Universal Robots PolyScope program: elton_fulltask.urp

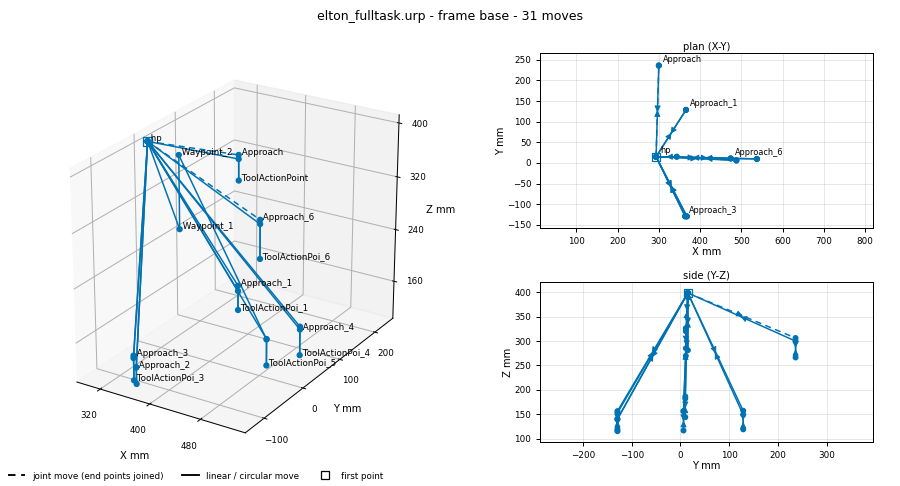
[picture p0: tool path of elton_fulltask.urp in frame base, 31 of 31 moves have a stored position in this frame; points joined in program order, loops and branches not executed]
Program elton_fulltask (installation=default directory=/programs createdIn=5.11.5.1010327 lastSavedIn=5.11.9.1010452 robotSerialNumber=20225200364)
Calibrated DH parameters: a=[0.00002, -0.569483, -0.54992, -0.00001, -0.000036, 0]; d=[0.180894, -146.691669, 192.918669, -46.053088, 0.119778, 0.115602]; alpha=[1.571425, -0.001534, 0.003359, 1.568739, -1.571477, 0]; deltaTheta=[0, 0.376258, -0.101074, -0.275185, -0.000002, 0]
Robot Program (runOnlyOnce=false)
  MoveL speed 250 mm/s, acceleration 1200 mm/s^2 (useActiveTCP=true) feature=Base
    Waypoint hp: TCP in base x=292.997 y=15.071 z=398.72 mm, rx=2.2312 ry=-2.2053 rz=0.0033 rad; joints [39.465, -75.549, -131.57, -243.154, -90.002, -141.049] deg
    URCap RG Grip (OnRobot, OnRobot A/S) dataModel(rg-target-force=40.0, rg-target-width=0.1)
    Loop Counting (count=6) loopVariable(name=Loop_2)
      URCap Palletizing (polyscope-pallet-impl, Universal Robots) dataModel(palletFeature=Base, isPalletizing=true, Length(key=objectHeight value=0.00001 unit=M), Variable(key=globalCountingVariable, variable(name=Pallet_4_cnt, initializeExpression=1)), Variable(key=layerNumberVariable, variable(name=Pallet_4_lno, initializeExpression=1)), Variable(key=layerCountingVariable, variable(name=Pallet_4_lct, initializeExpression=1)), Variable(key=handleSeparatorVariable, variable(name=Pallet_4_sep, initializeExpression=False)), Variable(key=totalCountVariable, variable(name=Pallet_4_tct, initializeExpression=1)), Variable(key=name, variable(name=R)), Variable(key=referencePoint, variable(featureName=referencePoin_3)), Variable(key=separatorPoint, variable(featureName=separatorPoin_3))); state(isChildrenLocked=true)
        URCap Patterns (polyscope-pallet-impl, Universal Robots) state(isChildrenLocked=true)
          URCap Pattern (polyscope-pallet-impl, Universal Robots) dataModel(UUID=4bae607c-6a0e-463c-838a-ad417c079e18, patternType=LINE, objects=6, Variable(key=nameVariable, variable(name=Line_Pattern_5))); state(isChildrenLocked=true)
            URCap Item (polyscope-pallet-impl, Universal Robots) dataModel(UUID=7363f219-9633-4242-9e50-65c058707edd, patternType=LINE, index=0, calibrationDeltaTheta=[-7.716858584048969E-7, 0.5809325624761351, 5.982441805008871, -0.2801932900558549, -2.087699179323388E-6, 7.182941588051994E-8], calibrationA=[5.584882619731399E-5, -0.5116748572506173, -0.549032347835167, 8.201669770320986E-5, -3.0447895639691726E-5, 0.0], calibrationD=[0.18058730552743416, -182.578946596082, 231.39006605348337, -48.6373829503458, 0.11974176219014578, 0.11553881708205978], calibrationAlpha=[1.5714381462339815, -0.001839843720035074, 0.003236774450590588, 1.5698364982897774, -1.571354041521518, 0.0], calibrationJointChecksum=[-1488423315, -1488334884, 658253144, -1490959501, -1490992896, -1492776484], calibrationStatus=2, calibrationValidChecksum=true, baseToFeature=[0.0, 0.0, 0.0, 0.0, 0.0, 0.0], TCPOffset=[-1.927819047531365E-5, -7.340324279514476E-6, -7.641604901187371E-6, 8.402270385809591E-6, 1.306011648505891E-6, 3.5749922966518936E-6], Variable(key=variable, variable(name=StartItem_5)), JointPositions(key=jointpositions, JointPosition(key=[1], Angle(key=pos value=1.151373 unit=RAD)), JointPosition(key=[2], Angle(key=pos value=-1.661465 unit=RAD)), JointPosition(key=[3], Angle(key=pos value=-2.268619 unit=RAD)), JointPosition(key=[4], Angle(key=pos value=-3.927088 unit=RAD)), JointPosition(key=[5], Angle(key=pos value=-1.572545 unit=RAD)), JointPosition(key=[6], Angle(key=pos value=-1.977698 unit=RAD))))
            URCap Item (polyscope-pallet-impl, Universal Robots) dataModel(UUID=34e06e1b-5aee-467a-bdea-27d33826544a, patternType=LINE, index=1, calibrationDeltaTheta=[-7.716858584048969E-7, 0.5809325624761351, 5.982441805008871, -0.2801932900558549, -2.087699179323388E-6, 7.182941588051994E-8], calibrationA=[5.584882619731399E-5, -0.5116748572506173, -0.549032347835167, 8.201669770320986E-5, -3.0447895639691726E-5, 0.0], calibrationD=[0.18058730552743416, -182.578946596082, 231.39006605348337, -48.6373829503458, 0.11974176219014578, 0.11553881708205978], calibrationAlpha=[1.5714381462339815, -0.001839843720035074, 0.003236774450590588, 1.5698364982897774, -1.571354041521518, 0.0], calibrationJointChecksum=[-1488423315, -1488334884, 658253144, -1490959501, -1490992896, -1492776484], calibrationStatus=2, calibrationValidChecksum=true, baseToFeature=[0.0, 0.0, 0.0, 0.0, 0.0, 0.0], TCPOffset=[-1.4484733942277117E-5, 2.1892267797196663E-6, -8.963613490398092E-6, 1.4148497921052897E-5, -4.324978428417448E-5, -3.9434016187655385E-5], Variable(key=variable, variable(name=EndItem_5)), JointPositions(key=jointpositions, JointPosition(key=[1], Angle(key=pos value=1.582831 unit=RAD)), JointPosition(key=[2], Angle(key=pos value=-1.495539 unit=RAD)), JointPosition(key=[3], Angle(key=pos value=-2.436687 unit=RAD)), JointPosition(key=[4], Angle(key=pos value=-3.925245 unit=RAD)), JointPosition(key=[5], Angle(key=pos value=-1.57402 unit=RAD)), JointPosition(key=[6], Angle(key=pos value=-1.546403 unit=RAD))))
        URCap Layers (polyscope-pallet-impl, Universal Robots) dataModel(separators=[false], selectedPatterns=[4bae607c-6a0e-463c-838a-ad417c079e18])
        URCap At Each Item (polyscope-pallet-impl, Universal Robots) dataModel(selectedPattern=4bae607c-6a0e-463c-838a-ad417c079e18, selectedPosition=7363f219-9633-4242-9e50-65c058707edd, Approach_calibrationDeltaTheta=[1.8465908720177726E-7, 0.2347954391419265, 6.32563174757166, -0.2772392005664852, -1.1261302130722607E-6, 2.5749233771577007E-7], Approach_calibrationA=[4.883734728215554E-5, -0.5955365338115801, -0.5495804852909227, 2.1882318399536237E-5, -4.077691201947169E-5, 0.0], Approach_calibrationD=[0.18075383087768818, -173.5375957069896, 228.42940994299985, -54.71797068756973, 0.11978402921182532, 0.11553172182396411], Approach_calibrationAlpha=[1.5713803919023464, -8.208946844426788E-4, 0.002849148556013, 1.569345144561223, -1.571367981038201, 0.0], Approach_calibrationJointChecksum=[-1454342380, -1456026624, 660707710, -1491716883, -1491592869, -1491595829], Approach_calibrationStatus=2, Approach_calibrationValidChecksum=true, Approach_baseToFeature=[0.0, 0.0, 0.0, 0.0, 0.0, 0.0], Approach_TCPOffset=[5.4603109008871664E-5, 2.376683340771235E-5, 1.3810152235949058E-5, -3.879481254340057E-5, 1.22456475810181E-4, -2.4036645708755116E-5], Exit_calibrationDeltaTheta=[1.8465908720177726E-7, 0.2347954391419265, 6.32563174757166, -0.2772392005664852, -1.1261302130722607E-6, 2.5749233771577007E-7], Exit_calibrationA=[4.883734728215554E-5, -0.5955365338115801, -0.5495804852909227, 2.1882318399536237E-5, -4.077691201947169E-5, 0.0], Exit_calibrationD=[0.18075383087768818, -173.5375957069896, 228.42940994299985, -54.71797068756973, 0.11978402921182532, 0.11553172182396411], Exit_calibrationAlpha=[1.5713803919023464, -8.208946844426788E-4, 0.002849148556013, 1.569345144561223, -1.571367981038201, 0.0], Exit_calibrationJointChecksum=[-1454342380, -1456026624, 660707710, -1491716883, -1491592869, -1491595829], Exit_calibrationStatus=2, Exit_calibrationValidChecksum=true, Exit_baseToFeature=[0.0, 0.0, 0.0, 0.0, 0.0, 0.0], Exit_TCPOffset=[5.458817584649833E-5, 2.1432463847392835E-5, 7.349381505572516E-5, -1.2814573171777247E-4, 1.0172603500468313E-4, -1.732072415206431E-5], currentWizardState=LANDING, Pose(key=refBaseToFeature, Position(key=posePosition, Length(key=X value=0 unit=M), Length(key=Y value=0 unit=M), Length(key=Z value=0 unit=M)), Rotation(key=poseRotation, Angle(key=RX value=0 unit=RAD), Angle(key=RY value=0 unit=RAD), Angle(key=RZ value=0 unit=RAD))), Pose(key=refPose, Position(key=posePosition, Length(key=X value=0.299651 unit=M), Length(key=Y value=0.236166 unit=M), Length(key=Z value=0.266297 unit=M)), Rotation(key=poseRotation, Angle(key=RX value=2.247176 unit=RAD), Angle(key=RY value=-2.190564 unit=RAD), Angle(key=RZ value=0.005192 unit=RAD))), JointPositions(key=Approach_jointpositions, JointPosition(key=[1], Angle(key=pos value=1.142609 unit=RAD)), JointPosition(key=[2], Angle(key=pos value=-1.611972 unit=RAD)), JointPosition(key=[3], Angle(key=pos value=-2.237967 unit=RAD)), JointPosition(key=[4], Angle(key=pos value=-4.008917 unit=RAD)), JointPosition(key=[5], Angle(key=pos value=-1.570991 unit=RAD)), JointPosition(key=[6], Angle(key=pos value=-2.021054 unit=RAD))), JointPositions(key=Exit_jointpositions, JointPosition(key=[1], Angle(key=pos value=1.142618 unit=RAD)), JointPosition(key=[2], Angle(key=pos value=-1.620563 unit=RAD)), JointPosition(key=[3], Angle(key=pos value=-2.243419 unit=RAD)), JointPosition(key=[4], Angle(key=pos value=-3.994874 unit=RAD)), JointPosition(key=[5], Angle(key=pos value=-1.570968 unit=RAD)), JointPosition(key=[6], Angle(key=pos value=-2.021008 unit=RAD))))
          URCap Generated Movements (polyscope-pallet-impl, Universal Robots) state(isChildrenLocked=true)
            MoveJ speed 60 deg/s, acceleration 80 deg/s^2 (useActiveTCP=true) feature=referencePoin_3
              Waypoint Approach: TCP in base x=299.628 y=236.111 z=306.226 mm, rx=2.2471 ry=-2.1905 rz=0.0053 rad; joints [65.467, -92.357, -128.232, -229.697, -90.01, -115.799] deg; TCP offset x=0 y=0 z=0 mm, rx=0 ry=0 rz=0 rad; feature pose in base x=299.651 y=236.166 z=266.297 mm, rx=2.2472 ry=-2.1906 rz=0.0052 rad
            MoveL speed 250 mm/s, acceleration 1200 mm/s^2 (useActiveTCP=true) feature(featureName=referencePoin_3)
              Waypoint ToolActionPoint: TCP in base x=299.651 y=236.166 z=266.297 mm, rx=2.2472 ry=-2.1906 rz=0.0052 rad; joints [65.47, -95.65, -130.086, -224.543, -90.002, -115.781] deg; TCP offset x=0 y=0 z=0 mm, rx=0 ry=0 rz=0 rad
            Folder Tool action
              URCap RG Grip (OnRobot, OnRobot A/S) dataModel(rg-target-force=40.0, rg-target-width=0.073)
            MoveL speed 250 mm/s, acceleration 1200 mm/s^2 (useActiveTCP=true) feature(featureName=referencePoin_3)
              Waypoint Exit_1: TCP in base x=299.631 y=236.111 z=299.866 mm, rx=2.2471 ry=-2.1904 rz=0.0052 rad; joints [65.465, -92.855, -128.546, -228.886, -90.014, -115.798] deg; TCP offset x=0 y=0 z=0 mm, rx=0 ry=0 rz=0 rad
      Waypoint hp: TCP in base x=292.997 y=15.071 z=398.72 mm, rx=2.2312 ry=-2.2053 rz=0.0033 rad; joints [39.465, -75.549, -131.57, -243.154, -90.002, -141.049] deg
      URCap Palletizing (polyscope-pallet-impl, Universal Robots) dataModel(palletFeature=Base, isPalletizing=true, Length(key=objectHeight value=0.00001 unit=M), Variable(key=globalCountingVariable, variable(name=Pallet_5_cnt, initializeExpression=1)), Variable(key=layerNumberVariable, variable(name=Pallet_5_lno, initializeExpression=1)), Variable(key=layerCountingVariable, variable(name=Pallet_5_lct, initializeExpression=1)), Variable(key=handleSeparatorVariable, variable(name=Pallet_5_sep, initializeExpression=False)), Variable(key=totalCountVariable, variable(name=Pallet_5_tct, initializeExpression=1)), Variable(key=name, variable(name=R2M)), Variable(key=referencePoint, variable(featureName=referencePoin_4)), Variable(key=separatorPoint, variable(featureName=separatorPoin_4))); state(isChildrenLocked=true)
        URCap Patterns (polyscope-pallet-impl, Universal Robots) state(isChildrenLocked=true)
          URCap Pattern (polyscope-pallet-impl, Universal Robots) dataModel(UUID=9dad8569-719f-4788-8023-540e95adebd7, patternType=LINE, objects=3, Variable(key=nameVariable, variable(name=Line_Pattern_6))); state(isChildrenLocked=true)
            URCap Item (polyscope-pallet-impl, Universal Robots) dataModel(UUID=9337c2a1-8eca-46a0-a6f6-7259e6f90a90, patternType=LINE, index=0, calibrationDeltaTheta=[-7.716858584048969E-7, 0.5809325624761351, 5.982441805008871, -0.2801932900558549, -2.087699179323388E-6, 7.182941588051994E-8], calibrationA=[5.584882619731399E-5, -0.5116748572506173, -0.549032347835167, 8.201669770320986E-5, -3.0447895639691726E-5, 0.0], calibrationD=[0.18058730552743416, -182.578946596082, 231.39006605348337, -48.6373829503458, 0.11974176219014578, 0.11553881708205978], calibrationAlpha=[1.5714381462339815, -0.001839843720035074, 0.003236774450590588, 1.5698364982897774, -1.571354041521518, 0.0], calibrationJointChecksum=[-1488423315, -1488334884, 658253144, -1490959501, -1490992896, -1492776484], calibrationStatus=2, calibrationValidChecksum=true, baseToFeature=[0.0, 0.0, 0.0, 0.0, 0.0, 0.0], TCPOffset=[7.065116085391843E-6, 6.19954151542812E-6, 1.9736858486663067E-5, -3.314970923571107E-5, 1.1768022558351274E-5, -4.2380350516320305E-5], Variable(key=variable, variable(name=StartItem_6)), JointPositions(key=jointpositions, JointPosition(key=[1], Angle(key=pos value=0.405971 unit=RAD)), JointPosition(key=[2], Angle(key=pos value=-1.817445 unit=RAD)), JointPosition(key=[3], Angle(key=pos value=-2.085999 unit=RAD)), JointPosition(key=[4], Angle(key=pos value=-3.952147 unit=RAD)), JointPosition(key=[5], Angle(key=pos value=-1.570877 unit=RAD)), JointPosition(key=[6], Angle(key=pos value=-2.723055 unit=RAD))))
            URCap Item (polyscope-pallet-impl, Universal Robots) dataModel(UUID=52735d64-6b3e-4983-aebc-b53ca12a7f6b, patternType=LINE, index=1, calibrationDeltaTheta=[-7.716858584048969E-7, 0.5809325624761351, 5.982441805008871, -0.2801932900558549, -2.087699179323388E-6, 7.182941588051994E-8], calibrationA=[5.584882619731399E-5, -0.5116748572506173, -0.549032347835167, 8.201669770320986E-5, -3.0447895639691726E-5, 0.0], calibrationD=[0.18058730552743416, -182.578946596082, 231.39006605348337, -48.6373829503458, 0.11974176219014578, 0.11553881708205978], calibrationAlpha=[1.5714381462339815, -0.001839843720035074, 0.003236774450590588, 1.5698364982897774, -1.571354041521518, 0.0], calibrationJointChecksum=[-1488423315, -1488334884, 658253144, -1490959501, -1490992896, -1492776484], calibrationStatus=2, calibrationValidChecksum=true, baseToFeature=[0.0, 0.0, 0.0, 0.0, 0.0, 0.0], TCPOffset=[-2.0043848415082083E-5, -7.908542197287982E-6, -1.8426994976394884E-5, 3.653735438177634E-5, -7.708839604067462E-5, -4.185073180004233E-5], Variable(key=variable, variable(name=EndItem_6)), JointPositions(key=jointpositions, JointPosition(key=[1], Angle(key=pos value=0.458346 unit=RAD)), JointPosition(key=[2], Angle(key=pos value=-1.739796 unit=RAD)), JointPosition(key=[3], Angle(key=pos value=-2.187725 unit=RAD)), JointPosition(key=[4], Angle(key=pos value=-3.928212 unit=RAD)), JointPosition(key=[5], Angle(key=pos value=-1.571032 unit=RAD)), JointPosition(key=[6], Angle(key=pos value=-2.670664 unit=RAD))))
          URCap Pattern (polyscope-pallet-impl, Universal Robots) dataModel(UUID=8783b59e-9459-45b0-8c56-a199d5abc192, patternType=LINE, objects=3, Variable(key=nameVariable, variable(name=Line_Pattern_7))); state(isChildrenLocked=true)
            URCap Item (polyscope-pallet-impl, Universal Robots) dataModel(UUID=6e9fca8b-d3fb-4757-91c2-e353f4d5e9d6, patternType=LINE, index=0, calibrationDeltaTheta=[-7.716858584048969E-7, 0.5809325624761351, 5.982441805008871, -0.2801932900558549, -2.087699179323388E-6, 7.182941588051994E-8], calibrationA=[5.584882619731399E-5, -0.5116748572506173, -0.549032347835167, 8.201669770320986E-5, -3.0447895639691726E-5, 0.0], calibrationD=[0.18058730552743416, -182.578946596082, 231.39006605348337, -48.6373829503458, 0.11974176219014578, 0.11553881708205978], calibrationAlpha=[1.5714381462339815, -0.001839843720035074, 0.003236774450590588, 1.5698364982897774, -1.571354041521518, 0.0], calibrationJointChecksum=[-1488423315, -1488334884, 658253144, -1490959501, -1490992896, -1492776484], calibrationStatus=2, calibrationValidChecksum=true, baseToFeature=[0.0, 0.0, 0.0, 0.0, 0.0, 0.0], TCPOffset=[1.256540876348744E-6, 4.99927723198422E-6, 1.0739034681572779E-5, -9.064806678141208E-6, 1.3852190798402818E-5, 3.6876369731935474E-5], Variable(key=variable, variable(name=StartItem_7)), JointPositions(key=jointpositions, JointPosition(key=[1], Angle(key=pos value=0.374591 unit=RAD)), JointPosition(key=[2], Angle(key=pos value=-1.75582 unit=RAD)), JointPosition(key=[3], Angle(key=pos value=-2.130395 unit=RAD)), JointPosition(key=[4], Angle(key=pos value=-3.965532 unit=RAD)), JointPosition(key=[5], Angle(key=pos value=-1.572848 unit=RAD)), JointPosition(key=[6], Angle(key=pos value=-4.345097 unit=RAD))))
            URCap Item (polyscope-pallet-impl, Universal Robots) dataModel(UUID=c0f000dd-f460-4563-86a8-3415e9775929, patternType=LINE, index=1, calibrationDeltaTheta=[-7.716858584048969E-7, 0.5809325624761351, 5.982441805008871, -0.2801932900558549, -2.087699179323388E-6, 7.182941588051994E-8], calibrationA=[5.584882619731399E-5, -0.5116748572506173, -0.549032347835167, 8.201669770320986E-5, -3.0447895639691726E-5, 0.0], calibrationD=[0.18058730552743416, -182.578946596082, 231.39006605348337, -48.6373829503458, 0.11974176219014578, 0.11553881708205978], calibrationAlpha=[1.5714381462339815, -0.001839843720035074, 0.003236774450590588, 1.5698364982897774, -1.571354041521518, 0.0], calibrationJointChecksum=[-1488423315, -1488334884, 658253144, -1490959501, -1490992896, -1492776484], calibrationStatus=2, calibrationValidChecksum=true, baseToFeature=[0.0, 0.0, 0.0, 0.0, 0.0, 0.0], TCPOffset=[7.74507941786462E-6, 1.410541287459599E-6, -1.2552769589502244E-5, 5.216667475077681E-5, 1.7428096929677165E-5, -7.606374204391279E-6], Variable(key=variable, variable(name=EndItem_7)), JointPositions(key=jointpositions, JointPosition(key=[1], Angle(key=pos value=0.488665 unit=RAD)), JointPosition(key=[2], Angle(key=pos value=-1.758563 unit=RAD)), JointPosition(key=[3], Angle(key=pos value=-2.126921 unit=RAD)), JointPosition(key=[4], Angle(key=pos value=-3.966372 unit=RAD)), JointPosition(key=[5], Angle(key=pos value=-1.572523 unit=RAD)), JointPosition(key=[6], Angle(key=pos value=-4.230996 unit=RAD))))
        URCap Layers (polyscope-pallet-impl, Universal Robots) dataModel(separators=[false, false], selectedPatterns=[9dad8569-719f-4788-8023-540e95adebd7, 8783b59e-9459-45b0-8c56-a199d5abc192])
        URCap At Each Item (polyscope-pallet-impl, Universal Robots) dataModel(selectedPattern=9dad8569-719f-4788-8023-540e95adebd7, selectedPosition=9337c2a1-8eca-46a0-a6f6-7259e6f90a90, Approach_calibrationDeltaTheta=[1.8465908720177726E-7, 0.2347954391419265, 6.32563174757166, -0.2772392005664852, -1.1261302130722607E-6, 2.5749233771577007E-7], Approach_calibrationA=[4.883734728215554E-5, -0.5955365338115801, -0.5495804852909227, 2.1882318399536237E-5, -4.077691201947169E-5, 0.0], Approach_calibrationD=[0.18075383087768818, -173.5375957069896, 228.42940994299985, -54.71797068756973, 0.11978402921182532, 0.11553172182396411], Approach_calibrationAlpha=[1.5713803919023464, -8.208946844426788E-4, 0.002849148556013, 1.569345144561223, -1.571367981038201, 0.0], Approach_calibrationJointChecksum=[-1454342380, -1456026624, 660707710, -1491716883, -1491592869, -1491595829], Approach_calibrationStatus=2, Approach_calibrationValidChecksum=true, Approach_baseToFeature=[0.0, 0.0, 0.0, 0.0, 0.0, 0.0], Approach_TCPOffset=[3.0238281606294846E-6, 1.2885141158880398E-5, 2.272453159168908E-5, -2.427481330974057E-5, 2.8413110607570904E-5, -3.767633446047109E-5], Exit_calibrationDeltaTheta=[1.8465908720177726E-7, 0.2347954391419265, 6.32563174757166, -0.2772392005664852, -1.1261302130722607E-6, 2.5749233771577007E-7], Exit_calibrationA=[4.883734728215554E-5, -0.5955365338115801, -0.5495804852909227, 2.1882318399536237E-5, -4.077691201947169E-5, 0.0], Exit_calibrationD=[0.18075383087768818, -173.5375957069896, 228.42940994299985, -54.71797068756973, 0.11978402921182532, 0.11553172182396411], Exit_calibrationAlpha=[1.5713803919023464, -8.208946844426788E-4, 0.002849148556013, 1.569345144561223, -1.571367981038201, 0.0], Exit_calibrationJointChecksum=[-1454342380, -1456026624, 660707710, -1491716883, -1491592869, -1491595829], Exit_calibrationStatus=2, Exit_calibrationValidChecksum=true, Exit_baseToFeature=[0.0, 0.0, 0.0, 0.0, 0.0, 0.0], Exit_TCPOffset=[-1.0906427108961243E-5, -1.1109997106850678E-5, 5.9044553536447E-6, 2.8945906654440277E-5, -1.2488270032187806E-5, -5.133849862661928E-5], currentWizardState=LANDING, Pose(key=refBaseToFeature, Position(key=posePosition, Length(key=X value=0 unit=M), Length(key=Y value=0 unit=M), Length(key=Z value=0 unit=M)), Rotation(key=poseRotation, Angle(key=RX value=0 unit=RAD), Angle(key=RY value=0 unit=RAD), Angle(key=RZ value=0 unit=RAD))), Pose(key=refPose, Position(key=posePosition, Length(key=X value=0.473862 unit=M), Length(key=Y value=0.010948 unit=M), Length(key=Z value=0.269628 unit=M)), Rotation(key=poseRotation, Angle(key=RX value=2.247173 unit=RAD), Angle(key=RY value=-2.190521 unit=RAD), Angle(key=RZ value=0.005152 unit=RAD))), JointPositions(key=Approach_jointpositions, JointPosition(key=[1], Angle(key=pos value=0.400666 unit=RAD)), JointPosition(key=[2], Angle(key=pos value=-1.740271 unit=RAD)), JointPosition(key=[3], Angle(key=pos value=-2.045306 unit=RAD)), JointPosition(key=[4], Angle(key=pos value=-4.070862 unit=RAD)), JointPosition(key=[5], Angle(key=pos value=-1.56858 unit=RAD)), JointPosition(key=[6], Angle(key=pos value=-2.763165 unit=RAD))), JointPositions(key=Exit_jointpositions, JointPosition(key=[1], Angle(key=pos value=0.40067 unit=RAD)), JointPosition(key=[2], Angle(key=pos value=-1.747145 unit=RAD)), JointPosition(key=[3], Angle(key=pos value=-2.050441 unit=RAD)), JointPosition(key=[4], Angle(key=pos value=-4.058853 unit=RAD)), JointPosition(key=[5], Angle(key=pos value=-1.568562 unit=RAD)), JointPosition(key=[6], Angle(key=pos value=-2.763129 unit=RAD))))
          URCap Generated Movements (polyscope-pallet-impl, Universal Robots) state(isChildrenLocked=true)
            MoveJ speed 60 deg/s, acceleration 80 deg/s^2 (useActiveTCP=true) feature=referencePoin_4
              Waypoint Approach_6: TCP in base x=473.849 y=10.945 z=326.348 mm, rx=2.2472 ry=-2.1905 rz=0.0052 rad; joints [22.957, -99.711, -117.19, -233.242, -89.872, -158.319] deg; TCP offset x=0 y=0 z=0 mm, rx=0 ry=0 rz=0 rad; feature pose in base x=473.862 y=10.948 z=269.628 mm, rx=2.2472 ry=-2.1905 rz=0.0052 rad
            MoveL speed 250 mm/s, acceleration 1200 mm/s^2 (useActiveTCP=true) feature(featureName=referencePoin_4)
              Waypoint ToolActionPoi_6: TCP in base x=473.862 y=10.948 z=269.628 mm, rx=2.2472 ry=-2.1905 rz=0.0052 rad; joints [22.958, -103.59, -119.645, -226.906, -89.862, -158.299] deg; TCP offset x=0 y=0 z=0 mm, rx=0 ry=0 rz=0 rad
            Folder Tool action
              URCap RG Grip (OnRobot, OnRobot A/S) dataModel(rg-target-force=40.0, rg-target-width=0.1)
            MoveL speed 250 mm/s, acceleration 1200 mm/s^2 (useActiveTCP=true) feature(featureName=referencePoin_4)
              Waypoint Exit_7: TCP in base x=473.873 y=10.959 z=320.174 mm, rx=2.2473 ry=-2.1905 rz=0.0052 rad; joints [22.957, -100.105, -117.481, -232.553, -89.872, -158.318] deg; TCP offset x=0 y=0 z=0 mm, rx=0 ry=0 rz=0 rad
    Waypoint hp: TCP in base x=292.997 y=15.071 z=398.72 mm, rx=2.2312 ry=-2.2053 rz=0.0033 rad; joints [39.465, -75.549, -131.57, -243.154, -90.002, -141.049] deg
    Loop Counting (count=6) loopVariable(name=Loop_3)
      URCap Palletizing (polyscope-pallet-impl, Universal Robots) dataModel(palletFeature=Base, isPalletizing=true, Length(key=objectHeight value=0.00001 unit=M), Variable(key=globalCountingVariable, variable(name=Pallet_6_cnt, initializeExpression=1)), Variable(key=layerNumberVariable, variable(name=Pallet_6_lno, initializeExpression=1)), Variable(key=layerCountingVariable, variable(name=Pallet_6_lct, initializeExpression=1)), Variable(key=handleSeparatorVariable, variable(name=Pallet_6_sep, initializeExpression=False)), Variable(key=totalCountVariable, variable(name=Pallet_6_tct, initializeExpression=1)), Variable(key=name, variable(name=L)), Variable(key=referencePoint, variable(featureName=referencePoin_5)), Variable(key=separatorPoint, variable(featureName=separatorPoin_5))); state(isChildrenLocked=true)
        URCap Patterns (polyscope-pallet-impl, Universal Robots) state(isChildrenLocked=true)
          URCap Pattern (polyscope-pallet-impl, Universal Robots) dataModel(UUID=4bae607c-6a0e-463c-838a-ad417c079e18, patternType=LINE, objects=6, Variable(key=nameVariable, variable(name=Line_Pattern_8))); state(isChildrenLocked=true)
            URCap Item (polyscope-pallet-impl, Universal Robots) dataModel(UUID=7363f219-9633-4242-9e50-65c058707edd, patternType=LINE, index=0, calibrationDeltaTheta=[-7.716858584048969E-7, 0.5809325624761351, 5.982441805008871, -0.2801932900558549, -2.087699179323388E-6, 7.182941588051994E-8], calibrationA=[5.584882619731399E-5, -0.5116748572506173, -0.549032347835167, 8.201669770320986E-5, -3.0447895639691726E-5, 0.0], calibrationD=[0.18058730552743416, -182.578946596082, 231.39006605348337, -48.6373829503458, 0.11974176219014578, 0.11553881708205978], calibrationAlpha=[1.5714381462339815, -0.001839843720035074, 0.003236774450590588, 1.5698364982897774, -1.571354041521518, 0.0], calibrationJointChecksum=[-1488423315, -1488334884, 658253144, -1490959501, -1490992896, -1492776484], calibrationStatus=2, calibrationValidChecksum=true, baseToFeature=[0.0, 0.0, 0.0, 0.0, 0.0, 0.0], TCPOffset=[-8.742061120697864E-6, 9.818390622751139E-6, -4.38230873689438E-6, -4.6643860458297756E-8, -2.0695401019555837E-5, -1.549763875015771E-5], Variable(key=variable, variable(name=StartItem_8)), JointPositions(key=jointpositions, JointPosition(key=[1], Angle(key=pos value=-0.120097 unit=RAD)), JointPosition(key=[2], Angle(key=pos value=-1.636462 unit=RAD)), JointPosition(key=[3], Angle(key=pos value=-2.295613 unit=RAD)), JointPosition(key=[4], Angle(key=pos value=-3.921959 unit=RAD)), JointPosition(key=[5], Angle(key=pos value=-1.571834 unit=RAD)), JointPosition(key=[6], Angle(key=pos value=-3.264863 unit=RAD))))
            URCap Item (polyscope-pallet-impl, Universal Robots) dataModel(UUID=34e06e1b-5aee-467a-bdea-27d33826544a, patternType=LINE, index=1, calibrationDeltaTheta=[-7.716858584048969E-7, 0.5809325624761351, 5.982441805008871, -0.2801932900558549, -2.087699179323388E-6, 7.182941588051994E-8], calibrationA=[5.584882619731399E-5, -0.5116748572506173, -0.549032347835167, 8.201669770320986E-5, -3.0447895639691726E-5, 0.0], calibrationD=[0.18058730552743416, -182.578946596082, 231.39006605348337, -48.6373829503458, 0.11974176219014578, 0.11553881708205978], calibrationAlpha=[1.5714381462339815, -0.001839843720035074, 0.003236774450590588, 1.5698364982897774, -1.571354041521518, 0.0], calibrationJointChecksum=[-1488423315, -1488334884, 658253144, -1490959501, -1490992896, -1492776484], calibrationStatus=2, calibrationValidChecksum=true, baseToFeature=[0.0, 0.0, 0.0, 0.0, 0.0, 0.0], TCPOffset=[3.359826186766224E-6, -4.265620550891747E-6, -2.207983904878308E-6, 6.176592076397044E-5, 3.0131039417098427E-5, -2.9922574415084677E-5], Variable(key=variable, variable(name=EndItem_8)), JointPositions(key=jointpositions, JointPosition(key=[1], Angle(key=pos value=-0.193527 unit=RAD)), JointPosition(key=[2], Angle(key=pos value=-1.447448 unit=RAD)), JointPosition(key=[3], Angle(key=pos value=-2.476456 unit=RAD)), JointPosition(key=[4], Angle(key=pos value=-3.929979 unit=RAD)), JointPosition(key=[5], Angle(key=pos value=-1.572174 unit=RAD)), JointPosition(key=[6], Angle(key=pos value=-3.338515 unit=RAD))))
        URCap Layers (polyscope-pallet-impl, Universal Robots) dataModel(separators=[false], selectedPatterns=[4bae607c-6a0e-463c-838a-ad417c079e18])
        URCap At Each Item (polyscope-pallet-impl, Universal Robots) dataModel(selectedPattern=4bae607c-6a0e-463c-838a-ad417c079e18, selectedPosition=7363f219-9633-4242-9e50-65c058707edd, Approach_calibrationDeltaTheta=[3.116151702300951E-8, 1.4166449605851306, 4.865070095092713, 0.0014795719880187595, -4.990860781074746E-7, -3.925871878279752E-8], Approach_calibrationA=[-1.0158439173703436E-5, -0.09403205366486023, -0.5713346358199152, 7.365520588418577E-5, -1.1425881794166018E-5, 0.0], Approach_calibrationD=[0.18077228301924886, -690.9574877576223, 691.0028500066884, 0.1288669073149633, 0.11969523249799581, 0.11554795361036506], Approach_calibrationAlpha=[1.5706246585230048, -8.758013512070892E-4, -0.018461075569511088, 1.5700128373526983, -1.56996879375117, 0.0], Approach_calibrationJointChecksum=[-1491211115, -1489904062, 825637646, -1324252155, -1324589245, -1493743004], Approach_calibrationStatus=2, Approach_calibrationValidChecksum=true, Approach_baseToFeature=[0.0, 0.0, 0.0, 0.0, 0.0, 0.0], Approach_TCPOffset=[-6.971843405978451E-6, -4.997208836177158E-7, -1.955075423698549E-5, -1.0986371840293002E-5, -5.911660278585862E-5, 4.719053038551945E-6], Exit_calibrationDeltaTheta=[3.116151702300951E-8, 1.4166449605851306, 4.865070095092713, 0.0014795719880187595, -4.990860781074746E-7, -3.925871878279752E-8], Exit_calibrationA=[-1.0158439173703436E-5, -0.09403205366486023, -0.5713346358199152, 7.365520588418577E-5, -1.1425881794166018E-5, 0.0], Exit_calibrationD=[0.18077228301924886, -690.9574877576223, 691.0028500066884, 0.1288669073149633, 0.11969523249799581, 0.11554795361036506], Exit_calibrationAlpha=[1.5706246585230048, -8.758013512070892E-4, -0.018461075569511088, 1.5700128373526983, -1.56996879375117, 0.0], Exit_calibrationJointChecksum=[-1491211115, -1489904062, 825637646, -1324252155, -1324589245, -1493743004], Exit_calibrationStatus=2, Exit_calibrationValidChecksum=true, Exit_baseToFeature=[0.0, 0.0, 0.0, 0.0, 0.0, 0.0], Exit_TCPOffset=[-2.883756055241382E-6, -8.764058286320209E-5, 6.748845653681279E-5, 2.233173570540951E-4, 1.0718237859408094E-7, -3.053486336395973E-5], currentWizardState=LANDING, Pose(key=refBaseToFeature, Position(key=posePosition, Length(key=X value=0 unit=M), Length(key=Y value=0 unit=M), Length(key=Z value=0 unit=M)), Rotation(key=poseRotation, Angle(key=RX value=0 unit=RAD), Angle(key=RY value=0 unit=RAD), Angle(key=RZ value=0 unit=RAD))), Pose(key=refPose, Position(key=posePosition, Length(key=X value=0.363576 unit=M), Length(key=Y value=-0.12936 unit=M), Length(key=Z value=0.119379 unit=M)), Rotation(key=poseRotation, Angle(key=RX value=-2.220753 unit=RAD), Angle(key=RY value=-2.19989 unit=RAD), Angle(key=RZ value=-0.045262 unit=RAD))), JointPositions(key=Approach_jointpositions, JointPosition(key=[1], Angle(key=pos value=0.111383 unit=RAD)), JointPosition(key=[2], Angle(key=pos value=-1.864744 unit=RAD)), JointPosition(key=[3], Angle(key=pos value=-2.314496 unit=RAD)), JointPosition(key=[4], Angle(key=pos value=2.622049 unit=RAD)), JointPosition(key=[5], Angle(key=pos value=-1.592615 unit=RAD)), JointPosition(key=[6], Angle(key=pos value=0.106175 unit=RAD))), JointPositions(key=Exit_jointpositions, JointPosition(key=[1], Angle(key=pos value=0.111362 unit=RAD)), JointPosition(key=[2], Angle(key=pos value=-1.871704 unit=RAD)), JointPosition(key=[3], Angle(key=pos value=-2.315767 unit=RAD)), JointPosition(key=[4], Angle(key=pos value=2.630276 unit=RAD)), JointPosition(key=[5], Angle(key=pos value=-1.592744 unit=RAD)), JointPosition(key=[6], Angle(key=pos value=0.106085 unit=RAD))))
          URCap Generated Movements (polyscope-pallet-impl, Universal Robots) state(isChildrenLocked=true)
            MoveL speed 250 mm/s, acceleration 1200 mm/s^2 (useActiveTCP=true) feature=referencePoin_5
              Waypoint Approach_3: TCP in base x=363.575 y=-129.368 z=156.241 mm, rx=-2.2208 ry=-2.1999 rz=-0.0452 rad; joints [6.382, -106.84, -132.611, 150.23, -91.247, 6.084] deg; TCP offset x=0 y=0 z=0 mm, rx=0 ry=0 rz=0 rad; feature pose in base x=363.576 y=-129.36 z=119.379 mm, rx=-2.2208 ry=-2.1999 rz=-0.0453 rad
            MoveL speed 250 mm/s, acceleration 1200 mm/s^2 (useActiveTCP=true) feature(featureName=referencePoin_5)
              Waypoint ToolActionPoi_3: TCP in base x=363.576 y=-129.36 z=119.379 mm, rx=-2.2208 ry=-2.1999 rz=-0.0453 rad; joints [6.371, -111.028, -133.222, 155.028, -91.327, 6.035] deg; TCP offset x=0 y=0 z=0 mm, rx=0 ry=0 rz=0 rad
            Folder Tool action
              URCap RG Grip (OnRobot, OnRobot A/S) dataModel(rg-target-force=40.0, rg-target-width=0.073)
            MoveL speed 250 mm/s, acceleration 1200 mm/s^2 (useActiveTCP=true) feature(featureName=referencePoin_5)
              Waypoint Exit_4: TCP in base x=363.489 y=-129.36 z=152.553 mm, rx=-2.2206 ry=-2.1998 rz=-0.045 rad; joints [6.382, -107.247, -132.692, 150.706, -91.259, 6.077] deg; TCP offset x=0 y=0 z=0 mm, rx=0 ry=0 rz=0 rad
      Waypoint hp: TCP in base x=292.997 y=15.071 z=398.72 mm, rx=2.2312 ry=-2.2053 rz=0.0033 rad; joints [39.465, -75.549, -131.57, -243.154, -90.002, -141.049] deg
      URCap Palletizing (polyscope-pallet-impl, Universal Robots) dataModel(palletFeature=Base, isPalletizing=true, Length(key=objectHeight value=0.00001 unit=M), Variable(key=name, variable(name=Pallet_7)), Variable(key=globalCountingVariable, variable(name=Pallet_7_cnt, initializeExpression=1)), Variable(key=layerNumberVariable, variable(name=Pallet_7_lno, initializeExpression=1)), Variable(key=layerCountingVariable, variable(name=Pallet_7_lct, initializeExpression=1)), Variable(key=handleSeparatorVariable, variable(name=Pallet_7_sep, initializeExpression=False)), Variable(key=totalCountVariable, variable(name=Pallet_7_tct, initializeExpression=1)), Variable(key=referencePoint, variable(featureName=referencePoin_6)), Variable(key=separatorPoint, variable(featureName=separatorPoin_6))); state(isChildrenLocked=true)
        URCap Patterns (polyscope-pallet-impl, Universal Robots) state(isChildrenLocked=true)
          URCap Pattern (polyscope-pallet-impl, Universal Robots) dataModel(UUID=9dad8569-719f-4788-8023-540e95adebd7, patternType=LINE, objects=3, Variable(key=nameVariable, variable(name=Line_Pattern_9))); state(isChildrenLocked=true)
            URCap Item (polyscope-pallet-impl, Universal Robots) dataModel(UUID=9337c2a1-8eca-46a0-a6f6-7259e6f90a90, patternType=LINE, index=0, calibrationDeltaTheta=[-2.1094217540068572E-7, 0.37625772532806073, -0.10107441100396769, -0.2751850025766889, -1.8024952768980196E-6, 2.9402326063437956E-8], calibrationA=[2.0416891277915125E-5, -0.5694828868469309, -0.5499202125525207, -9.504674691390763E-6, -3.603723657207661E-5, 0.0], calibrationD=[0.1808937726775539, -146.69166934821124, 192.91866861971778, -46.05308757405963, 0.11977780403821288, 0.11560212559305974], calibrationAlpha=[1.5714252480212174, -0.0015337665762078037, 0.0033588312559612306, 1.5687392298942362, -1.5714772428732047, 0.0], calibrationJointChecksum=[-1490546360, -1456574554, -1506622700, -1493399207, -1492840923, -1492940558], calibrationStatus=2, calibrationValidChecksum=true, baseToFeature=[0.0, 0.0, 0.0, 0.0, 0.0, 0.0], TCPOffset=[-9.784447780127742E-6, 2.6810172487068407E-6, 7.281711053797046E-6, -1.989125181765513E-6, -1.364623003286183E-5, -4.713350057546712E-6], Variable(key=variable, variable(name=StartItem_9)), JointPositions(key=jointpositions, JointPosition(key=[1], Angle(key=pos value=0.401157 unit=RAD)), JointPosition(key=[2], Angle(key=pos value=-1.784677 unit=RAD)), JointPosition(key=[3], Angle(key=pos value=-2.058624 unit=RAD)), JointPosition(key=[4], Angle(key=pos value=-4.011941 unit=RAD)), JointPosition(key=[5], Angle(key=pos value=-1.571492 unit=RAD)), JointPosition(key=[6], Angle(key=pos value=-2.742725 unit=RAD))))
            URCap Item (polyscope-pallet-impl, Universal Robots) dataModel(UUID=52735d64-6b3e-4983-aebc-b53ca12a7f6b, patternType=LINE, index=1, calibrationDeltaTheta=[-2.1094217540068572E-7, 0.37625772532806073, -0.10107441100396769, -0.2751850025766889, -1.8024952768980196E-6, 2.9402326063437956E-8], calibrationA=[2.0416891277915125E-5, -0.5694828868469309, -0.5499202125525207, -9.504674691390763E-6, -3.603723657207661E-5, 0.0], calibrationD=[0.1808937726775539, -146.69166934821124, 192.91866861971778, -46.05308757405963, 0.11977780403821288, 0.11560212559305974], calibrationAlpha=[1.5714252480212174, -0.0015337665762078037, 0.0033588312559612306, 1.5687392298942362, -1.5714772428732047, 0.0], calibrationJointChecksum=[-1490546360, -1456574554, -1506622700, -1493399207, -1492840923, -1492940558], calibrationStatus=2, calibrationValidChecksum=true, baseToFeature=[0.0, 0.0, 0.0, 0.0, 0.0, 0.0], TCPOffset=[-2.6756666668056872E-5, 3.2672035924496967E-6, 1.5707032072265203E-5, -1.5722457421381595E-5, 2.2020802890041943E-5, -3.831152369534655E-5], Variable(key=variable, variable(name=EndItem_9)), JointPositions(key=jointpositions, JointPosition(key=[1], Angle(key=pos value=0.451425 unit=RAD)), JointPosition(key=[2], Angle(key=pos value=-1.702339 unit=RAD)), JointPosition(key=[3], Angle(key=pos value=-2.161102 unit=RAD)), JointPosition(key=[4], Angle(key=pos value=-3.991986 unit=RAD)), JointPosition(key=[5], Angle(key=pos value=-1.571567 unit=RAD)), JointPosition(key=[6], Angle(key=pos value=-2.692565 unit=RAD))))
          URCap Pattern (polyscope-pallet-impl, Universal Robots) dataModel(UUID=8783b59e-9459-45b0-8c56-a199d5abc192, patternType=LINE, objects=3, Variable(key=nameVariable, variable(name=Line_Pattern_10))); state(isChildrenLocked=true)
            URCap Item (polyscope-pallet-impl, Universal Robots) dataModel(UUID=6e9fca8b-d3fb-4757-91c2-e353f4d5e9d6, patternType=LINE, index=0, calibrationDeltaTheta=[-2.1094217540068572E-7, 0.37625772532806073, -0.10107441100396769, -0.2751850025766889, -1.8024952768980196E-6, 2.9402326063437956E-8], calibrationA=[2.0416891277915125E-5, -0.5694828868469309, -0.5499202125525207, -9.504674691390763E-6, -3.603723657207661E-5, 0.0], calibrationD=[0.1808937726775539, -146.69166934821124, 192.91866861971778, -46.05308757405963, 0.11977780403821288, 0.11560212559305974], calibrationAlpha=[1.5714252480212174, -0.0015337665762078037, 0.0033588312559612306, 1.5687392298942362, -1.5714772428732047, 0.0], calibrationJointChecksum=[-1490546360, -1456574554, -1506622700, -1493399207, -1492840923, -1492940558], calibrationStatus=2, calibrationValidChecksum=true, baseToFeature=[0.0, 0.0, 0.0, 0.0, 0.0, 0.0], TCPOffset=[-2.030488224780136E-7, -1.3789832864982005E-5, -1.114379750494221E-5, -7.008563005896843E-6, 4.953911986066089E-5, -9.035229078160812E-5], Variable(key=variable, variable(name=StartItem_10)), JointPositions(key=jointpositions, JointPosition(key=[1], Angle(key=pos value=0.361911 unit=RAD)), JointPosition(key=[2], Angle(key=pos value=-1.726918 unit=RAD)), JointPosition(key=[3], Angle(key=pos value=-2.10642 unit=RAD)), JointPosition(key=[4], Angle(key=pos value=-4.019181 unit=RAD)), JointPosition(key=[5], Angle(key=pos value=-1.573128 unit=RAD)), JointPosition(key=[6], Angle(key=pos value=-4.375697 unit=RAD))))
            URCap Item (polyscope-pallet-impl, Universal Robots) dataModel(UUID=c0f000dd-f460-4563-86a8-3415e9775929, patternType=LINE, index=1, calibrationDeltaTheta=[-2.1094217540068572E-7, 0.37625772532806073, -0.10107441100396769, -0.2751850025766889, -1.8024952768980196E-6, 2.9402326063437956E-8], calibrationA=[2.0416891277915125E-5, -0.5694828868469309, -0.5499202125525207, -9.504674691390763E-6, -3.603723657207661E-5, 0.0], calibrationD=[0.1808937726775539, -146.69166934821124, 192.91866861971778, -46.05308757405963, 0.11977780403821288, 0.11560212559305974], calibrationAlpha=[1.5714252480212174, -0.0015337665762078037, 0.0033588312559612306, 1.5687392298942362, -1.5714772428732047, 0.0], calibrationJointChecksum=[-1490546360, -1456574554, -1506622700, -1493399207, -1492840923, -1492940558], calibrationStatus=2, calibrationValidChecksum=true, baseToFeature=[0.0, 0.0, 0.0, 0.0, 0.0, 0.0], TCPOffset=[-1.0971008582549846E-5, 1.104955046919709E-5, 1.5323638876629797E-5, -1.6494841423695708E-5, -3.927198589300623E-5, -1.0718793121454852E-5], Variable(key=variable, variable(name=EndItem_10)), JointPositions(key=jointpositions, JointPosition(key=[1], Angle(key=pos value=0.490255 unit=RAD)), JointPosition(key=[2], Angle(key=pos value=-1.719243 unit=RAD)), JointPosition(key=[3], Angle(key=pos value=-2.107888 unit=RAD)), JointPosition(key=[4], Angle(key=pos value=-4.02554 unit=RAD)), JointPosition(key=[5], Angle(key=pos value=-1.572902 unit=RAD)), JointPosition(key=[6], Angle(key=pos value=-4.24229 unit=RAD))))
        URCap Layers (polyscope-pallet-impl, Universal Robots) dataModel(separators=[false, false], selectedPatterns=[9dad8569-719f-4788-8023-540e95adebd7, 8783b59e-9459-45b0-8c56-a199d5abc192])
        URCap At Each Item (polyscope-pallet-impl, Universal Robots) dataModel(selectedPattern=9dad8569-719f-4788-8023-540e95adebd7, selectedPosition=9337c2a1-8eca-46a0-a6f6-7259e6f90a90, Approach_calibrationDeltaTheta=[3.116151702300951E-8, 1.4166449605851306, 4.865070095092713, 0.0014795719880187595, -4.990860781074746E-7, -3.925871878279752E-8], Approach_calibrationA=[-1.0158439173703436E-5, -0.09403205366486023, -0.5713346358199152, 7.365520588418577E-5, -1.1425881794166018E-5, 0.0], Approach_calibrationD=[0.18077228301924886, -690.9574877576223, 691.0028500066884, 0.1288669073149633, 0.11969523249799581, 0.11554795361036506], Approach_calibrationAlpha=[1.5706246585230048, -8.758013512070892E-4, -0.018461075569511088, 1.5700128373526983, -1.56996879375117, 0.0], Approach_calibrationJointChecksum=[-1491211115, -1489904062, 825637646, -1324252155, -1324589245, -1493743004], Approach_calibrationStatus=2, Approach_calibrationValidChecksum=true, Approach_baseToFeature=[0.0, 0.0, 0.0, 0.0, 0.0, 0.0], Approach_TCPOffset=[4.708636894359269E-6, -1.1802683406170189E-5, 3.0890270187156066E-5, 3.469685434437999E-5, -5.936535457447061E-5, -4.4645763785282684E-5], Exit_calibrationDeltaTheta=[3.116151702300951E-8, 1.4166449605851306, 4.865070095092713, 0.0014795719880187595, -4.990860781074746E-7, -3.925871878279752E-8], Exit_calibrationA=[-1.0158439173703436E-5, -0.09403205366486023, -0.5713346358199152, 7.365520588418577E-5, -1.1425881794166018E-5, 0.0], Exit_calibrationD=[0.18077228301924886, -690.9574877576223, 691.0028500066884, 0.1288669073149633, 0.11969523249799581, 0.11554795361036506], Exit_calibrationAlpha=[1.5706246585230048, -8.758013512070892E-4, -0.018461075569511088, 1.5700128373526983, -1.56996879375117, 0.0], Exit_calibrationJointChecksum=[-1491211115, -1489904062, 825637646, -1324252155, -1324589245, -1493743004], Exit_calibrationStatus=2, Exit_calibrationValidChecksum=true, Exit_baseToFeature=[0.0, 0.0, 0.0, 0.0, 0.0, 0.0], Exit_TCPOffset=[9.940978031384995E-6, -1.317045104154424E-5, -4.763215142256083E-6, 2.445351077417118E-5, 4.019062692039104E-6, -2.1499032796649547E-5], currentWizardState=LANDING, Pose(key=refBaseToFeature, Position(key=posePosition, Length(key=X value=0 unit=M), Length(key=Y value=0 unit=M), Length(key=Z value=0 unit=M)), Rotation(key=poseRotation, Angle(key=RX value=0 unit=RAD), Angle(key=RY value=0 unit=RAD), Angle(key=RZ value=0 unit=RAD))), Pose(key=refPose, Position(key=posePosition, Length(key=X value=0.53743 unit=M), Length(key=Y value=0.009852 unit=M), Length(key=Z value=0.143758 unit=M)), Rotation(key=poseRotation, Angle(key=RX value=2.228407 unit=RAD), Angle(key=RY value=2.206337 unit=RAD), Angle(key=RZ value=-0.001996 unit=RAD))), JointPositions(key=Approach_jointpositions, JointPosition(key=[1], Angle(key=pos value=0.346393 unit=RAD)), JointPosition(key=[2], Angle(key=pos value=-2.010305 unit=RAD)), JointPosition(key=[3], Angle(key=pos value=-1.997183 unit=RAD)), JointPosition(key=[4], Angle(key=pos value=2.438894 unit=RAD)), JointPosition(key=[5], Angle(key=pos value=-1.55405 unit=RAD)), JointPosition(key=[6], Angle(key=pos value=0.343508 unit=RAD))), JointPositions(key=Exit_jointpositions, JointPosition(key=[1], Angle(key=pos value=0.34641 unit=RAD)), JointPosition(key=[2], Angle(key=pos value=-2.004407 unit=RAD)), JointPosition(key=[3], Angle(key=pos value=-1.995576 unit=RAD)), JointPosition(key=[4], Angle(key=pos value=2.431389 unit=RAD)), JointPosition(key=[5], Angle(key=pos value=-1.553948 unit=RAD)), JointPosition(key=[6], Angle(key=pos value=0.343611 unit=RAD))))
          URCap Generated Movements (polyscope-pallet-impl, Universal Robots) state(isChildrenLocked=true)
            MoveL speed 250 mm/s, acceleration 1200 mm/s^2 (useActiveTCP=true) feature=referencePoin_6
              Waypoint Approach_4: TCP in base x=537.419 y=9.856 z=181.969 mm, rx=2.2283 ry=2.2064 rz=-0.0021 rad; joints [19.848, -115.184, -114.432, 139.739, -89.038, 19.681] deg; TCP offset x=0 y=0 z=0 mm, rx=0 ry=0 rz=0 rad; feature pose in base x=537.43 y=9.852 z=143.758 mm, rx=2.2284 ry=2.2063 rz=-0.002 rad
            MoveL speed 250 mm/s, acceleration 1200 mm/s^2 (useActiveTCP=true) feature(featureName=referencePoin_6)
              Waypoint ToolActionPoi_4: TCP in base x=537.43 y=9.852 z=143.758 mm, rx=2.2284 ry=2.2063 rz=-0.002 rad; joints [19.839, -118.289, -115.105, 143.52, -89.094, 19.632] deg; TCP offset x=0 y=0 z=0 mm, rx=0 ry=0 rz=0 rad
            Folder Tool action
              URCap RG Grip (OnRobot, OnRobot A/S) dataModel(rg-target-force=40.0, rg-target-width=0.1)
            MoveL speed 250 mm/s, acceleration 1200 mm/s^2 (useActiveTCP=true) feature(featureName=referencePoin_6)
              Waypoint Exit_5: TCP in base x=537.417 y=9.862 z=186.305 mm, rx=2.2284 ry=2.2064 rz=-0.002 rad; joints [19.849, -114.843, -114.339, 139.307, -89.035, 19.688] deg; TCP offset x=0 y=0 z=0 mm, rx=0 ry=0 rz=0 rad
  MoveL speed 250 mm/s, acceleration 1200 mm/s^2 (useActiveTCP=true) feature=Base
    Waypoint hp: TCP in base x=292.997 y=15.071 z=398.72 mm, rx=2.2312 ry=-2.2053 rz=0.0033 rad; joints [39.465, -75.549, -131.57, -243.154, -90.002, -141.049] deg
    URCap RG Grip (OnRobot, OnRobot A/S) dataModel(rg-target-force=40.0, rg-target-width=0.1, Variable(key=on_return, variable(name=on_return)))
    Loop Counting (count=12) loopVariable(name=Loop_1)
      URCap Palletizing (polyscope-pallet-impl, Universal Robots) dataModel(palletFeature=Base, isPalletizing=false, Variable(key=name, variable(name=Pallet_1)), Variable(key=globalCountingVariable, variable(name=Pallet_1_cnt_1, initializeExpression=1)), Variable(key=layerNumberVariable, variable(name=Pallet_1_lno, initializeExpression=1)), Variable(key=layerCountingVariable, variable(name=Pallet_1_lct, initializeExpression=1)), Variable(key=handleSeparatorVariable, variable(name=Pallet_1_sep, initializeExpression=False)), Variable(key=totalCountVariable, variable(name=Pallet_1_tct, initializeExpression=1)), Length(key=objectHeight value=0.00001 unit=M), Variable(key=referencePoint, variable(featureName=referencePoint)), Variable(key=separatorPoint, variable(featureName=separatorPoint))); state(isChildrenLocked=true)
        URCap Patterns (polyscope-pallet-impl, Universal Robots) state(isChildrenLocked=true)
          URCap Pattern (polyscope-pallet-impl, Universal Robots) dataModel(UUID=29e288a1-ce4c-47a2-9416-0f60e082fc2d, patternType=LINE, objects=3, Variable(key=nameVariable, variable(name=floor4))); state(isChildrenLocked=true)
            URCap Item (polyscope-pallet-impl, Universal Robots) dataModel(UUID=00e49389-8ad2-43e5-99dc-a8ec89804c66, patternType=LINE, index=0, calibrationDeltaTheta=[-7.716858584048969E-7, 0.5809325624761351, 5.982441805008871, -0.2801932900558549, -2.087699179323388E-6, 7.182941588051994E-8], calibrationA=[5.584882619731399E-5, -0.5116748572506173, -0.549032347835167, 8.201669770320986E-5, -3.0447895639691726E-5, 0.0], calibrationD=[0.18058730552743416, -182.578946596082, 231.39006605348337, -48.6373829503458, 0.11974176219014578, 0.11553881708205978], calibrationAlpha=[1.5714381462339815, -0.001839843720035074, 0.003236774450590588, 1.5698364982897774, -1.571354041521518, 0.0], calibrationJointChecksum=[-1488423315, -1488334884, 658253144, -1490959501, -1490992896, -1492776484], calibrationStatus=2, calibrationValidChecksum=true, baseToFeature=[0.0, 0.0, 0.0, 0.0, 0.0, 0.0], TCPOffset=[-1.300925221525695E-5, -4.503482033249573E-6, 2.1768893027240832E-5, -2.9392173756652047E-5, -5.2383955626649044E-5, -2.0115477830749817E-5], Variable(key=variable, variable(name=StartItem_1)), JointPositions(key=jointpositions, JointPosition(key=[1], Angle(key=pos value=0.479524 unit=RAD)), JointPosition(key=[2], Angle(key=pos value=-1.722598 unit=RAD)), JointPosition(key=[3], Angle(key=pos value=-2.100361 unit=RAD)), JointPosition(key=[4], Angle(key=pos value=-4.029606 unit=RAD)), JointPosition(key=[5], Angle(key=pos value=-1.57312 unit=RAD)), JointPosition(key=[6], Angle(key=pos value=-4.213238 unit=RAD))))
            URCap Item (polyscope-pallet-impl, Universal Robots) dataModel(UUID=a0c7d3d6-1887-4a88-b7d3-44a22bc40ae2, patternType=LINE, index=1, calibrationDeltaTheta=[-7.716858584048969E-7, 0.5809325624761351, 5.982441805008871, -0.2801932900558549, -2.087699179323388E-6, 7.182941588051994E-8], calibrationA=[5.584882619731399E-5, -0.5116748572506173, -0.549032347835167, 8.201669770320986E-5, -3.0447895639691726E-5, 0.0], calibrationD=[0.18058730552743416, -182.578946596082, 231.39006605348337, -48.6373829503458, 0.11974176219014578, 0.11553881708205978], calibrationAlpha=[1.5714381462339815, -0.001839843720035074, 0.003236774450590588, 1.5698364982897774, -1.571354041521518, 0.0], calibrationJointChecksum=[-1488423315, -1488334884, 658253144, -1490959501, -1490992896, -1492776484], calibrationStatus=2, calibrationValidChecksum=true, baseToFeature=[0.0, 0.0, 0.0, 0.0, 0.0, 0.0], TCPOffset=[1.3476539566181778E-5, -1.451539108707732E-5, -2.551666819244902E-5, 2.145716645190336E-5, 1.8494716812647057E-5, 1.1939568656688123E-5], Variable(key=variable, variable(name=EndItem_1)), JointPositions(key=jointpositions, JointPosition(key=[1], Angle(key=pos value=0.37183 unit=RAD)), JointPosition(key=[2], Angle(key=pos value=-1.720273 unit=RAD)), JointPosition(key=[3], Angle(key=pos value=-2.103233 unit=RAD)), JointPosition(key=[4], Angle(key=pos value=-4.029064 unit=RAD)), JointPosition(key=[5], Angle(key=pos value=-1.573299 unit=RAD)), JointPosition(key=[6], Angle(key=pos value=-4.320966 unit=RAD))))
          URCap Pattern (polyscope-pallet-impl, Universal Robots) dataModel(UUID=277ca75e-475c-4893-88be-ec8a720a9350, patternType=LINE, objects=3, Variable(key=nameVariable, variable(name=Line_Pattern_4))); state(isChildrenLocked=true)
            URCap Item (polyscope-pallet-impl, Universal Robots) dataModel(UUID=24e8ef12-c2c6-4028-b23d-237b5cb4d535, patternType=LINE, index=0, calibrationDeltaTheta=[-7.716858584048969E-7, 0.5809325624761351, 5.982441805008871, -0.2801932900558549, -2.087699179323388E-6, 7.182941588051994E-8], calibrationA=[5.584882619731399E-5, -0.5116748572506173, -0.549032347835167, 8.201669770320986E-5, -3.0447895639691726E-5, 0.0], calibrationD=[0.18058730552743416, -182.578946596082, 231.39006605348337, -48.6373829503458, 0.11974176219014578, 0.11553881708205978], calibrationAlpha=[1.5714381462339815, -0.001839843720035074, 0.003236774450590588, 1.5698364982897774, -1.571354041521518, 0.0], calibrationJointChecksum=[-1488423315, -1488334884, 658253144, -1490959501, -1490992896, -1492776484], calibrationStatus=2, calibrationValidChecksum=true, baseToFeature=[0.0, 0.0, 0.0, 0.0, 0.0, 0.0], TCPOffset=[-6.537227036168547E-6, 8.123743144350382E-6, -1.8023699240865554E-6, -1.2017156694174843E-5, -2.1693669029424024E-5, 1.1742333824028037E-5], Variable(key=variable, variable(name=StartItem_4)), JointPositions(key=jointpositions, JointPosition(key=[1], Angle(key=pos value=0.452837 unit=RAD)), JointPosition(key=[2], Angle(key=pos value=-1.698611 unit=RAD)), JointPosition(key=[3], Angle(key=pos value=-2.164495 unit=RAD)), JointPosition(key=[4], Angle(key=pos value=-3.992209 unit=RAD)), JointPosition(key=[5], Angle(key=pos value=-1.57189 unit=RAD)), JointPosition(key=[6], Angle(key=pos value=-2.692104 unit=RAD))))
            URCap Item (polyscope-pallet-impl, Universal Robots) dataModel(UUID=f0f9be9e-3032-48e0-bc89-15ff320ca791, patternType=LINE, index=1, calibrationDeltaTheta=[-7.716858584048969E-7, 0.5809325624761351, 5.982441805008871, -0.2801932900558549, -2.087699179323388E-6, 7.182941588051994E-8], calibrationA=[5.584882619731399E-5, -0.5116748572506173, -0.549032347835167, 8.201669770320986E-5, -3.0447895639691726E-5, 0.0], calibrationD=[0.18058730552743416, -182.578946596082, 231.39006605348337, -48.6373829503458, 0.11974176219014578, 0.11553881708205978], calibrationAlpha=[1.5714381462339815, -0.001839843720035074, 0.003236774450590588, 1.5698364982897774, -1.571354041521518, 0.0], calibrationJointChecksum=[-1488423315, -1488334884, 658253144, -1490959501, -1490992896, -1492776484], calibrationStatus=2, calibrationValidChecksum=true, baseToFeature=[0.0, 0.0, 0.0, 0.0, 0.0, 0.0], TCPOffset=[1.2641931620959931E-5, 5.139564874412361E-6, 2.0700093662506802E-5, -5.9922875285412244E-5, 2.9797049357115657E-5, 1.328717889618731E-5], Variable(key=variable, variable(name=EndItem_4)), JointPositions(key=jointpositions, JointPosition(key=[1], Angle(key=pos value=0.403821 unit=RAD)), JointPosition(key=[2], Angle(key=pos value=-1.778608 unit=RAD)), JointPosition(key=[3], Angle(key=pos value=-2.065516 unit=RAD)), JointPosition(key=[4], Angle(key=pos value=-4.011076 unit=RAD)), JointPosition(key=[5], Angle(key=pos value=-1.571783 unit=RAD)), JointPosition(key=[6], Angle(key=pos value=-2.741098 unit=RAD))))
          URCap Pattern (polyscope-pallet-impl, Universal Robots) dataModel(UUID=cad00631-a279-4055-bdc3-ca350480e51d, patternType=LINE, objects=3, Variable(key=nameVariable, variable(name=Line_Pattern_11))); state(isChildrenLocked=true)
            URCap Item (polyscope-pallet-impl, Universal Robots) dataModel(UUID=8ea465ab-a401-4b4f-b9c8-e012120d6ab5, patternType=LINE, index=0, calibrationDeltaTheta=[-7.716858584048969E-7, 0.5809325624761351, 5.982441805008871, -0.2801932900558549, -2.087699179323388E-6, 7.182941588051994E-8], calibrationA=[5.584882619731399E-5, -0.5116748572506173, -0.549032347835167, 8.201669770320986E-5, -3.0447895639691726E-5, 0.0], calibrationD=[0.18058730552743416, -182.578946596082, 231.39006605348337, -48.6373829503458, 0.11974176219014578, 0.11553881708205978], calibrationAlpha=[1.5714381462339815, -0.001839843720035074, 0.003236774450590588, 1.5698364982897774, -1.571354041521518, 0.0], calibrationJointChecksum=[-1488423315, -1488334884, 658253144, -1490959501, -1490992896, -1492776484], calibrationStatus=2, calibrationValidChecksum=true, baseToFeature=[0.0, 0.0, 0.0, 0.0, 0.0, 0.0], TCPOffset=[-2.101063999976338E-5, 2.586532609974261E-5, 2.4885786296391377E-5, -8.926250995045922E-5, -6.786156528647164E-5, 1.5797495797581828E-6], Variable(key=variable, variable(name=StartItem_11)), JointPositions(key=jointpositions, JointPosition(key=[1], Angle(key=pos value=0.374582 unit=RAD)), JointPosition(key=[2], Angle(key=pos value=-1.755832 unit=RAD)), JointPosition(key=[3], Angle(key=pos value=-2.130403 unit=RAD)), JointPosition(key=[4], Angle(key=pos value=-3.965503 unit=RAD)), JointPosition(key=[5], Angle(key=pos value=-1.572834 unit=RAD)), JointPosition(key=[6], Angle(key=pos value=-4.345068 unit=RAD))))
            URCap Item (polyscope-pallet-impl, Universal Robots) dataModel(UUID=a9157890-d2eb-469b-b8b0-703fba5bd283, patternType=LINE, index=1, calibrationDeltaTheta=[-7.716858584048969E-7, 0.5809325624761351, 5.982441805008871, -0.2801932900558549, -2.087699179323388E-6, 7.182941588051994E-8], calibrationA=[5.584882619731399E-5, -0.5116748572506173, -0.549032347835167, 8.201669770320986E-5, -3.0447895639691726E-5, 0.0], calibrationD=[0.18058730552743416, -182.578946596082, 231.39006605348337, -48.6373829503458, 0.11974176219014578, 0.11553881708205978], calibrationAlpha=[1.5714381462339815, -0.001839843720035074, 0.003236774450590588, 1.5698364982897774, -1.571354041521518, 0.0], calibrationJointChecksum=[-1488423315, -1488334884, 658253144, -1490959501, -1490992896, -1492776484], calibrationStatus=2, calibrationValidChecksum=true, baseToFeature=[0.0, 0.0, 0.0, 0.0, 0.0, 0.0], TCPOffset=[3.4129516318648356E-7, -9.94379794682504E-6, -8.703321898173577E-6, -3.814941872790498E-5, -9.35249682044337E-6, -2.448973663716019E-5], Variable(key=variable, variable(name=EndItem_11)), JointPositions(key=jointpositions, JointPosition(key=[1], Angle(key=pos value=0.488643 unit=RAD)), JointPosition(key=[2], Angle(key=pos value=-1.758548 unit=RAD)), JointPosition(key=[3], Angle(key=pos value=-2.126899 unit=RAD)), JointPosition(key=[4], Angle(key=pos value=-3.966369 unit=RAD)), JointPosition(key=[5], Angle(key=pos value=-1.572562 unit=RAD)), JointPosition(key=[6], Angle(key=pos value=-4.231026 unit=RAD))))
          URCap Pattern (polyscope-pallet-impl, Universal Robots) dataModel(UUID=f62da871-c8c3-4d57-adb7-a9a8a6b66379, patternType=LINE, objects=3, Variable(key=nameVariable, variable(name=Line_Pattern_12))); state(isChildrenLocked=true)
            URCap Item (polyscope-pallet-impl, Universal Robots) dataModel(UUID=cc5c7a7e-cff9-4b23-a2f9-b5a5d8978f72, patternType=LINE, index=0, calibrationDeltaTheta=[-7.716858584048969E-7, 0.5809325624761351, 5.982441805008871, -0.2801932900558549, -2.087699179323388E-6, 7.182941588051994E-8], calibrationA=[5.584882619731399E-5, -0.5116748572506173, -0.549032347835167, 8.201669770320986E-5, -3.0447895639691726E-5, 0.0], calibrationD=[0.18058730552743416, -182.578946596082, 231.39006605348337, -48.6373829503458, 0.11974176219014578, 0.11553881708205978], calibrationAlpha=[1.5714381462339815, -0.001839843720035074, 0.003236774450590588, 1.5698364982897774, -1.571354041521518, 0.0], calibrationJointChecksum=[-1488423315, -1488334884, 658253144, -1490959501, -1490992896, -1492776484], calibrationStatus=2, calibrationValidChecksum=true, baseToFeature=[0.0, 0.0, 0.0, 0.0, 0.0, 0.0], TCPOffset=[-1.6700120912465505E-5, 2.2963211916471327E-5, 2.4125457564083685E-5, -8.571297031944018E-5, 4.626318871520733E-5, -2.6696804905816887E-5], Variable(key=variable, variable(name=StartItem_12)), JointPositions(key=jointpositions, JointPosition(key=[1], Angle(key=pos value=0.405961 unit=RAD)), JointPosition(key=[2], Angle(key=pos value=-1.817472 unit=RAD)), JointPosition(key=[3], Angle(key=pos value=-2.08602 unit=RAD)), JointPosition(key=[4], Angle(key=pos value=-3.952135 unit=RAD)), JointPosition(key=[5], Angle(key=pos value=-1.570879 unit=RAD)), JointPosition(key=[6], Angle(key=pos value=-2.723107 unit=RAD))))
            URCap Item (polyscope-pallet-impl, Universal Robots) dataModel(UUID=b01a9c46-84f1-42ec-a875-d71a6fee28b6, patternType=LINE, index=1, calibrationDeltaTheta=[-7.716858584048969E-7, 0.5809325624761351, 5.982441805008871, -0.2801932900558549, -2.087699179323388E-6, 7.182941588051994E-8], calibrationA=[5.584882619731399E-5, -0.5116748572506173, -0.549032347835167, 8.201669770320986E-5, -3.0447895639691726E-5, 0.0], calibrationD=[0.18058730552743416, -182.578946596082, 231.39006605348337, -48.6373829503458, 0.11974176219014578, 0.11553881708205978], calibrationAlpha=[1.5714381462339815, -0.001839843720035074, 0.003236774450590588, 1.5698364982897774, -1.571354041521518, 0.0], calibrationJointChecksum=[-1488423315, -1488334884, 658253144, -1490959501, -1490992896, -1492776484], calibrationStatus=2, calibrationValidChecksum=true, baseToFeature=[0.0, 0.0, 0.0, 0.0, 0.0, 0.0], TCPOffset=[6.418304604478148E-6, -7.33343933395636E-6, 3.2820347403705874E-6, 2.864912960614694E-7, -3.550807467998849E-5, 3.418648131386808E-5], Variable(key=variable, variable(name=EndItem_12)), JointPositions(key=jointpositions, JointPosition(key=[1], Angle(key=pos value=0.458367 unit=RAD)), JointPosition(key=[2], Angle(key=pos value=-1.739765 unit=RAD)), JointPosition(key=[3], Angle(key=pos value=-2.187699 unit=RAD)), JointPosition(key=[4], Angle(key=pos value=-3.928202 unit=RAD)), JointPosition(key=[5], Angle(key=pos value=-1.571084 unit=RAD)), JointPosition(key=[6], Angle(key=pos value=-2.670685 unit=RAD))))
        URCap Layers (polyscope-pallet-impl, Universal Robots) dataModel(separators=[false, false, false, false], selectedPatterns=[f62da871-c8c3-4d57-adb7-a9a8a6b66379, cad00631-a279-4055-bdc3-ca350480e51d, 277ca75e-475c-4893-88be-ec8a720a9350, 29e288a1-ce4c-47a2-9416-0f60e082fc2d])
        URCap At Each Item (polyscope-pallet-impl, Universal Robots) dataModel(selectedPattern=29e288a1-ce4c-47a2-9416-0f60e082fc2d, selectedPosition=00e49389-8ad2-43e5-99dc-a8ec89804c66, Approach_calibrationDeltaTheta=[3.116151702300951E-8, 1.4166449605851306, 4.865070095092713, 0.0014795719880187595, -4.990860781074746E-7, -3.925871878279752E-8], Approach_calibrationA=[-1.0158439173703436E-5, -0.09403205366486023, -0.5713346358199152, 7.365520588418577E-5, -1.1425881794166018E-5, 0.0], Approach_calibrationD=[0.18077228301924886, -690.9574877576223, 691.0028500066884, 0.1288669073149633, 0.11969523249799581, 0.11554795361036506], Approach_calibrationAlpha=[1.5706246585230048, -8.758013512070892E-4, -0.018461075569511088, 1.5700128373526983, -1.56996879375117, 0.0], Approach_calibrationJointChecksum=[-1491211115, -1489904062, 825637646, -1324252155, -1324589245, -1493743004], Approach_calibrationStatus=2, Approach_calibrationValidChecksum=true, Approach_baseToFeature=[0.0, 0.0, 0.0, 0.0, 0.0, 0.0], Approach_TCPOffset=[-5.47743179733079E-7, 1.5218694433438706E-5, 2.611463367080402E-6, -3.811931631810776E-5, 2.0545972804589437E-6, 2.622779555432771E-5], Exit_calibrationDeltaTheta=[3.116151702300951E-8, 1.4166449605851306, 4.865070095092713, 0.0014795719880187595, -4.990860781074746E-7, -3.925871878279752E-8], Exit_calibrationA=[-1.0158439173703436E-5, -0.09403205366486023, -0.5713346358199152, 7.365520588418577E-5, -1.1425881794166018E-5, 0.0], Exit_calibrationD=[0.18077228301924886, -690.9574877576223, 691.0028500066884, 0.1288669073149633, 0.11969523249799581, 0.11554795361036506], Exit_calibrationAlpha=[1.5706246585230048, -8.758013512070892E-4, -0.018461075569511088, 1.5700128373526983, -1.56996879375117, 0.0], Exit_calibrationJointChecksum=[-1491211115, -1489904062, 825637646, -1324252155, -1324589245, -1493743004], Exit_calibrationStatus=2, Exit_calibrationValidChecksum=true, Exit_baseToFeature=[0.0, 0.0, 0.0, 0.0, 0.0, 0.0], Exit_TCPOffset=[-1.2260723835227916E-6, -2.3822357979430553E-5, 2.5240997519382358E-5, 4.590928010718624E-5, -2.4190326273446138E-5, -4.632519642109508E-6], currentWizardState=LANDING, Pose(key=refBaseToFeature, Position(key=posePosition, Length(key=X value=0 unit=M), Length(key=Y value=0 unit=M), Length(key=Z value=0 unit=M)), Rotation(key=poseRotation, Angle(key=RX value=0 unit=RAD), Angle(key=RY value=0 unit=RAD), Angle(key=RZ value=0 unit=RAD))), Pose(key=refPose, Position(key=posePosition, Length(key=X value=0.487642 unit=M), Length(key=Y value=0.006206 unit=M), Length(key=Z value=0.116442 unit=M)), Rotation(key=poseRotation, Angle(key=RX value=2.228217 unit=RAD), Angle(key=RY value=2.206466 unit=RAD), Angle(key=RZ value=-0.002174 unit=RAD))), JointPositions(key=Approach_jointpositions, JointPosition(key=[1], Angle(key=pos value=0.375678 unit=RAD)), JointPosition(key=[2], Angle(key=pos value=-1.988386 unit=RAD)), JointPosition(key=[3], Angle(key=pos value=-2.108921 unit=RAD)), JointPosition(key=[4], Angle(key=pos value=2.528462 unit=RAD)), JointPosition(key=[5], Angle(key=pos value=-1.555249 unit=RAD)), JointPosition(key=[6], Angle(key=pos value=0.371624 unit=RAD))), JointPositions(key=Exit_jointpositions, JointPosition(key=[1], Angle(key=pos value=0.375675 unit=RAD)), JointPosition(key=[2], Angle(key=pos value=-1.989328 unit=RAD)), JointPosition(key=[3], Angle(key=pos value=-2.109103 unit=RAD)), JointPosition(key=[4], Angle(key=pos value=2.529587 unit=RAD)), JointPosition(key=[5], Angle(key=pos value=-1.555266 unit=RAD)), JointPosition(key=[6], Angle(key=pos value=0.37161 unit=RAD))))
          URCap Generated Movements (polyscope-pallet-impl, Universal Robots) state(isChildrenLocked=true)
            MoveL speed 250 mm/s, acceleration 1200 mm/s^2 (useActiveTCP=true) feature=referencePoint
              Waypoint Approach_5: TCP in base x=487.657 y=6.206 z=156.384 mm, rx=2.2282 ry=2.2064 rz=-0.0021 rad; joints [21.524, -113.927, -120.831, 144.872, -89.109, 21.293] deg; TCP offset x=0 y=0 z=0 mm, rx=0 ry=0 rz=0 rad; feature pose in base x=487.642 y=6.206 z=116.442 mm, rx=2.2282 ry=2.2065 rz=-0.0022 rad
            MoveL speed 250 mm/s, acceleration 1200 mm/s^2 (useActiveTCP=true) feature(featureName=referencePoint)
              Waypoint ToolActionPoi_5: TCP in base x=487.642 y=6.206 z=116.442 mm, rx=2.2282 ry=2.2065 rz=-0.0022 rad; joints [21.516, -117.608, -121.377, 149.097, -89.173, 21.244] deg; TCP offset x=0 y=0 z=0 mm, rx=0 ry=0 rz=0 rad
            Folder Tool action
              URCap RG Grip (OnRobot, OnRobot A/S) dataModel(rg-target-force=40.0, rg-target-width=0.073)
            MoveL speed 250 mm/s, acceleration 1200 mm/s^2 (useActiveTCP=true) feature(featureName=referencePoint)
              Waypoint Exit_6: TCP in base x=487.618 y=6.205 z=155.759 mm, rx=2.2282 ry=2.2065 rz=-0.0023 rad; joints [21.526, -113.982, -120.845, 144.936, -89.11, 21.292] deg; TCP offset x=0 y=0 z=0 mm, rx=0 ry=0 rz=0 rad
      MoveL speed 250 mm/s, acceleration 1200 mm/s^2 (useActiveTCP=true) feature=Base
        Waypoint Waypoint_2: TCP in base x=343.195 y=15.137 z=389.494 mm, rx=2.2108 ry=-2.2293 rz=0.0032 rad; joints [33, -82.427, -127.279, -240.413, -90.075, -146.344] deg
        Waypoint Waypoint_1: TCP in base x=343.192 y=15.131 z=281.125 mm, rx=2.2107 ry=-2.2293 rz=0.0032 rad; joints [33.029, -90.394, -133.587, -226.14, -90.045, -146.262] deg
        Wait Sleep waitTime=1
        If analog_in[0]<5
          MoveL speed 250 mm/s, acceleration 1200 mm/s^2 (useActiveTCP=true) feature=Base
            Waypoint hp: TCP in base x=292.997 y=15.071 z=398.72 mm, rx=2.2312 ry=-2.2053 rz=0.0033 rad; joints [39.465, -75.549, -131.57, -243.154, -90.002, -141.049] deg
            URCap Palletizing (polyscope-pallet-impl, Universal Robots) dataModel(palletFeature=Base, isPalletizing=true, Variable(key=name, variable(name=Pallet_2)), Variable(key=globalCountingVariable, variable(name=Pallet_2_cnt, initializeExpression=1)), Variable(key=layerNumberVariable, variable(name=Pallet_2_lno, initializeExpression=1)), Variable(key=layerCountingVariable, variable(name=Pallet_2_lct, initializeExpression=1)), Variable(key=handleSeparatorVariable, variable(name=Pallet_2_sep, initializeExpression=False)), Variable(key=totalCountVariable, variable(name=Pallet_2_tct, initializeExpression=1)), Length(key=objectHeight value=0.00001 unit=M), Variable(key=referencePoint, variable(featureName=referencePoin_1)), Variable(key=separatorPoint, variable(featureName=separatorPoin_1))); state(isChildrenLocked=true)
              URCap Patterns (polyscope-pallet-impl, Universal Robots) state(isChildrenLocked=true)
                URCap Pattern (polyscope-pallet-impl, Universal Robots) dataModel(UUID=90a39d43-6053-4ac2-aa15-f126633cbd8f, patternType=LINE, objects=6, Variable(key=nameVariable, variable(name=Line_Pattern_2))); state(isChildrenLocked=true)
                  URCap Item (polyscope-pallet-impl, Universal Robots) dataModel(UUID=21ba8069-eb30-42b9-b937-0a2dd4e205a7, patternType=LINE, index=0, calibrationDeltaTheta=[-7.716858584048969E-7, 0.5809325624761351, 5.982441805008871, -0.2801932900558549, -2.087699179323388E-6, 7.182941588051994E-8], calibrationA=[5.584882619731399E-5, -0.5116748572506173, -0.549032347835167, 8.201669770320986E-5, -3.0447895639691726E-5, 0.0], calibrationD=[0.18058730552743416, -182.578946596082, 231.39006605348337, -48.6373829503458, 0.11974176219014578, 0.11553881708205978], calibrationAlpha=[1.5714381462339815, -0.001839843720035074, 0.003236774450590588, 1.5698364982897774, -1.571354041521518, 0.0], calibrationJointChecksum=[-1488423315, -1488334884, 658253144, -1490959501, -1490992896, -1492776484], calibrationStatus=2, calibrationValidChecksum=true, baseToFeature=[0.0, 0.0, 0.0, 0.0, 0.0, 0.0], TCPOffset=[-2.936942902709294E-6, 9.503995376941576E-6, 7.632028847792682E-6, -4.10927646012327E-5, 3.929885852369315E-5, -6.661916422680447E-5], Variable(key=variable, variable(name=StartItem_2)), JointPositions(key=jointpositions, JointPosition(key=[1], Angle(key=pos value=1.582846 unit=RAD)), JointPosition(key=[2], Angle(key=pos value=-1.495527 unit=RAD)), JointPosition(key=[3], Angle(key=pos value=-2.436664 unit=RAD)), JointPosition(key=[4], Angle(key=pos value=-3.925239 unit=RAD)), JointPosition(key=[5], Angle(key=pos value=-1.574005 unit=RAD)), JointPosition(key=[6], Angle(key=pos value=-1.546428 unit=RAD))))
                  URCap Item (polyscope-pallet-impl, Universal Robots) dataModel(UUID=d88c14ed-9ea8-4bbb-9d1f-9b7ce0149a47, patternType=LINE, index=1, calibrationDeltaTheta=[-7.716858584048969E-7, 0.5809325624761351, 5.982441805008871, -0.2801932900558549, -2.087699179323388E-6, 7.182941588051994E-8], calibrationA=[5.584882619731399E-5, -0.5116748572506173, -0.549032347835167, 8.201669770320986E-5, -3.0447895639691726E-5, 0.0], calibrationD=[0.18058730552743416, -182.578946596082, 231.39006605348337, -48.6373829503458, 0.11974176219014578, 0.11553881708205978], calibrationAlpha=[1.5714381462339815, -0.001839843720035074, 0.003236774450590588, 1.5698364982897774, -1.571354041521518, 0.0], calibrationJointChecksum=[-1488423315, -1488334884, 658253144, -1490959501, -1490992896, -1492776484], calibrationStatus=2, calibrationValidChecksum=true, baseToFeature=[0.0, 0.0, 0.0, 0.0, 0.0, 0.0], TCPOffset=[-2.5686336043551083E-5, 3.064455791845777E-6, -2.477735667133496E-5, 1.6339378998548308E-5, -8.85152565341253E-5, -3.277206579265757E-5], Variable(key=variable, variable(name=EndItem_2)), JointPositions(key=jointpositions, JointPosition(key=[1], Angle(key=pos value=1.151376 unit=RAD)), JointPosition(key=[2], Angle(key=pos value=-1.661484 unit=RAD)), JointPosition(key=[3], Angle(key=pos value=-2.268579 unit=RAD)), JointPosition(key=[4], Angle(key=pos value=-3.927109 unit=RAD)), JointPosition(key=[5], Angle(key=pos value=-1.572545 unit=RAD)), JointPosition(key=[6], Angle(key=pos value=-1.977695 unit=RAD))))
              URCap Layers (polyscope-pallet-impl, Universal Robots) dataModel(separators=[false], selectedPatterns=[90a39d43-6053-4ac2-aa15-f126633cbd8f])
              URCap At Each Item (polyscope-pallet-impl, Universal Robots) dataModel(selectedPattern=90a39d43-6053-4ac2-aa15-f126633cbd8f, selectedPosition=21ba8069-eb30-42b9-b937-0a2dd4e205a7, Approach_calibrationDeltaTheta=[3.116151702300951E-8, 1.4166449605851306, 4.865070095092713, 0.0014795719880187595, -4.990860781074746E-7, -3.925871878279752E-8], Approach_calibrationA=[-1.0158439173703436E-5, -0.09403205366486023, -0.5713346358199152, 7.365520588418577E-5, -1.1425881794166018E-5, 0.0], Approach_calibrationD=[0.18077228301924886, -690.9574877576223, 691.0028500066884, 0.1288669073149633, 0.11969523249799581, 0.11554795361036506], Approach_calibrationAlpha=[1.5706246585230048, -8.758013512070892E-4, -0.018461075569511088, 1.5700128373526983, -1.56996879375117, 0.0], Approach_calibrationJointChecksum=[-1491211115, -1489904062, 825637646, -1324252155, -1324589245, -1493743004], Approach_calibrationStatus=2, Approach_calibrationValidChecksum=true, Approach_baseToFeature=[0.0, 0.0, 0.0, 0.0, 0.0, 0.0], Approach_TCPOffset=[-1.5216007202611959E-5, 6.762418482075816E-6, 1.0126156336304204E-5, 3.423419794696584E-5, -4.128360146718241E-5, 1.8976382015290816E-5], Exit_calibrationDeltaTheta=[3.116151702300951E-8, 1.4166449605851306, 4.865070095092713, 0.0014795719880187595, -4.990860781074746E-7, -3.925871878279752E-8], Exit_calibrationA=[-1.0158439173703436E-5, -0.09403205366486023, -0.5713346358199152, 7.365520588418577E-5, -1.1425881794166018E-5, 0.0], Exit_calibrationD=[0.18077228301924886, -690.9574877576223, 691.0028500066884, 0.1288669073149633, 0.11969523249799581, 0.11554795361036506], Exit_calibrationAlpha=[1.5706246585230048, -8.758013512070892E-4, -0.018461075569511088, 1.5700128373526983, -1.56996879375117, 0.0], Exit_calibrationJointChecksum=[-1491211115, -1489904062, 825637646, -1324252155, -1324589245, -1493743004], Exit_calibrationStatus=2, Exit_calibrationValidChecksum=true, Exit_baseToFeature=[0.0, 0.0, 0.0, 0.0, 0.0, 0.0], Exit_TCPOffset=[-3.1161778783761473E-6, -2.2609839781584373E-5, 1.0672103324949056E-6, 4.8162794144324856E-5, -2.0027443108690995E-5, -7.779198954957423E-5], currentWizardState=LANDING, Pose(key=refBaseToFeature, Position(key=posePosition, Length(key=X value=0 unit=M), Length(key=Y value=0 unit=M), Length(key=Z value=0 unit=M)), Rotation(key=poseRotation, Angle(key=RX value=0 unit=RAD), Angle(key=RY value=0 unit=RAD), Angle(key=RZ value=0 unit=RAD))), Pose(key=refPose, Position(key=posePosition, Length(key=X value=0.365592 unit=M), Length(key=Y value=0.128732 unit=M), Length(key=Z value=0.118831 unit=M)), Rotation(key=poseRotation, Angle(key=RX value=2.228342 unit=RAD), Angle(key=RY value=2.206338 unit=RAD), Angle(key=RZ value=-0.001907 unit=RAD))), JointPositions(key=Approach_jointpositions, JointPosition(key=[1], Angle(key=pos value=0.801563 unit=RAD)), JointPosition(key=[2], Angle(key=pos value=-1.86812 unit=RAD)), JointPosition(key=[3], Angle(key=pos value=-2.312023 unit=RAD)), JointPosition(key=[4], Angle(key=pos value=2.608965 unit=RAD)), JointPosition(key=[5], Angle(key=pos value=-1.556657 unit=RAD)), JointPosition(key=[6], Angle(key=pos value=0.796733 unit=RAD))), JointPositions(key=Exit_jointpositions, JointPosition(key=[1], Angle(key=pos value=0.801515 unit=RAD)), JointPosition(key=[2], Angle(key=pos value=-1.884199 unit=RAD)), JointPosition(key=[3], Angle(key=pos value=-2.314843 unit=RAD)), JointPosition(key=[4], Angle(key=pos value=2.627864 unit=RAD)), JointPosition(key=[5], Angle(key=pos value=-1.556953 unit=RAD)), JointPosition(key=[6], Angle(key=pos value=0.796524 unit=RAD))))
                URCap Generated Movements (polyscope-pallet-impl, Universal Robots) state(isChildrenLocked=true)
                  MoveL speed 250 mm/s, acceleration 1200 mm/s^2 (useActiveTCP=true) feature=referencePoin_1
                    Waypoint Approach_1: TCP in base x=365.599 y=128.717 z=156.964 mm, rx=2.2284 ry=2.2063 rz=-0.002 rad; joints [45.924, -107.038, -132.469, 149.481, -89.19, 45.648] deg; TCP offset x=0 y=0 z=0 mm, rx=0 ry=0 rz=0 rad; feature pose in base x=365.592 y=128.732 z=118.831 mm, rx=2.2283 ry=2.2063 rz=-0.0019 rad
                  MoveL speed 250 mm/s, acceleration 1200 mm/s^2 (useActiveTCP=true) feature(featureName=referencePoin_1)
                    Waypoint ToolActionPoi_1: TCP in base x=365.592 y=128.732 z=118.831 mm, rx=2.2283 ry=2.2063 rz=-0.0019 rad; joints [45.914, -111.365, -133.087, 154.43, -89.269, 45.598] deg; TCP offset x=0 y=0 z=0 mm, rx=0 ry=0 rz=0 rad
                  Folder Tool action
                    URCap RG Grip (OnRobot, OnRobot A/S) dataModel(rg-target-force=40.0, rg-target-width=0.1)
                  MoveL speed 250 mm/s, acceleration 1200 mm/s^2 (useActiveTCP=true) feature(featureName=referencePoin_1)
                    Waypoint Exit_2: TCP in base x=365.57 y=128.729 z=148.673 mm, rx=2.2283 ry=2.2064 rz=-0.002 rad; joints [45.925, -107.956, -132.633, 150.564, -89.208, 45.635] deg; TCP offset x=0 y=0 z=0 mm, rx=0 ry=0 rz=0 rad
        Else 
          MoveL speed 250 mm/s, acceleration 1200 mm/s^2 (useActiveTCP=true) feature=Base
            Waypoint hp: TCP in base x=292.997 y=15.071 z=398.72 mm, rx=2.2312 ry=-2.2053 rz=0.0033 rad; joints [39.465, -75.549, -131.57, -243.154, -90.002, -141.049] deg
            URCap Palletizing (polyscope-pallet-impl, Universal Robots) dataModel(palletFeature=Base, isPalletizing=true, Length(key=objectHeight value=0.00001 unit=M), Variable(key=name, variable(name=Pallet_3)), Variable(key=globalCountingVariable, variable(name=Pallet_3_cnt, initializeExpression=1)), Variable(key=layerNumberVariable, variable(name=Pallet_3_lno, initializeExpression=1)), Variable(key=layerCountingVariable, variable(name=Pallet_3_lct, initializeExpression=1)), Variable(key=handleSeparatorVariable, variable(name=Pallet_3_sep, initializeExpression=False)), Variable(key=totalCountVariable, variable(name=Pallet_3_tct, initializeExpression=1)), Variable(key=referencePoint, variable(featureName=referencePoin_2)), Variable(key=separatorPoint, variable(featureName=separatorPoin_2))); state(isChildrenLocked=true)
              URCap Patterns (polyscope-pallet-impl, Universal Robots) state(isChildrenLocked=true)
                URCap Pattern (polyscope-pallet-impl, Universal Robots) dataModel(UUID=90a39d43-6053-4ac2-aa15-f126633cbd8f, patternType=LINE, objects=6, Variable(key=nameVariable, variable(name=Line_Pattern_3))); state(isChildrenLocked=true)
                  URCap Item (polyscope-pallet-impl, Universal Robots) dataModel(UUID=21ba8069-eb30-42b9-b937-0a2dd4e205a7, patternType=LINE, index=0, calibrationDeltaTheta=[-7.716858584048969E-7, 0.5809325624761351, 5.982441805008871, -0.2801932900558549, -2.087699179323388E-6, 7.182941588051994E-8], calibrationA=[5.584882619731399E-5, -0.5116748572506173, -0.549032347835167, 8.201669770320986E-5, -3.0447895639691726E-5, 0.0], calibrationD=[0.18058730552743416, -182.578946596082, 231.39006605348337, -48.6373829503458, 0.11974176219014578, 0.11553881708205978], calibrationAlpha=[1.5714381462339815, -0.001839843720035074, 0.003236774450590588, 1.5698364982897774, -1.571354041521518, 0.0], calibrationJointChecksum=[-1488423315, -1488334884, 658253144, -1490959501, -1490992896, -1492776484], calibrationStatus=2, calibrationValidChecksum=true, baseToFeature=[0.0, 0.0, 0.0, 0.0, 0.0, 0.0], TCPOffset=[6.167002582491143E-6, 1.3157397689478323E-5, -1.4073136301751E-5, 5.0848806525472837E-5, 9.43396056796775E-6, 5.0237808367789265E-5], Variable(key=variable, variable(name=StartItem_3)), JointPositions(key=jointpositions, JointPosition(key=[1], Angle(key=pos value=-0.193529 unit=RAD)), JointPosition(key=[2], Angle(key=pos value=-1.447425 unit=RAD)), JointPosition(key=[3], Angle(key=pos value=-2.47645 unit=RAD)), JointPosition(key=[4], Angle(key=pos value=-3.929942 unit=RAD)), JointPosition(key=[5], Angle(key=pos value=-1.572157 unit=RAD)), JointPosition(key=[6], Angle(key=pos value=-3.338547 unit=RAD))))
                  URCap Item (polyscope-pallet-impl, Universal Robots) dataModel(UUID=d88c14ed-9ea8-4bbb-9d1f-9b7ce0149a47, patternType=LINE, index=1, calibrationDeltaTheta=[-7.716858584048969E-7, 0.5809325624761351, 5.982441805008871, -0.2801932900558549, -2.087699179323388E-6, 7.182941588051994E-8], calibrationA=[5.584882619731399E-5, -0.5116748572506173, -0.549032347835167, 8.201669770320986E-5, -3.0447895639691726E-5, 0.0], calibrationD=[0.18058730552743416, -182.578946596082, 231.39006605348337, -48.6373829503458, 0.11974176219014578, 0.11553881708205978], calibrationAlpha=[1.5714381462339815, -0.001839843720035074, 0.003236774450590588, 1.5698364982897774, -1.571354041521518, 0.0], calibrationJointChecksum=[-1488423315, -1488334884, 658253144, -1490959501, -1490992896, -1492776484], calibrationStatus=2, calibrationValidChecksum=true, baseToFeature=[0.0, 0.0, 0.0, 0.0, 0.0, 0.0], TCPOffset=[5.739068194093866E-6, 1.2249660714724886E-5, 1.8669901249435128E-5, -8.520564219610992E-5, -1.8506468913075373E-5, -2.827152451905457E-5], Variable(key=variable, variable(name=EndItem_3)), JointPositions(key=jointpositions, JointPosition(key=[1], Angle(key=pos value=-0.120081 unit=RAD)), JointPosition(key=[2], Angle(key=pos value=-1.636435 unit=RAD)), JointPosition(key=[3], Angle(key=pos value=-2.295632 unit=RAD)), JointPosition(key=[4], Angle(key=pos value=-3.921969 unit=RAD)), JointPosition(key=[5], Angle(key=pos value=-1.571855 unit=RAD)), JointPosition(key=[6], Angle(key=pos value=-3.264862 unit=RAD))))
              URCap Layers (polyscope-pallet-impl, Universal Robots) dataModel(separators=[false], selectedPatterns=[90a39d43-6053-4ac2-aa15-f126633cbd8f])
              URCap At Each Item (polyscope-pallet-impl, Universal Robots) dataModel(selectedPattern=90a39d43-6053-4ac2-aa15-f126633cbd8f, selectedPosition=21ba8069-eb30-42b9-b937-0a2dd4e205a7, Approach_calibrationDeltaTheta=[3.116151702300951E-8, 1.4166449605851306, 4.865070095092713, 0.0014795719880187595, -4.990860781074746E-7, -3.925871878279752E-8], Approach_calibrationA=[-1.0158439173703436E-5, -0.09403205366486023, -0.5713346358199152, 7.365520588418577E-5, -1.1425881794166018E-5, 0.0], Approach_calibrationD=[0.18077228301924886, -690.9574877576223, 691.0028500066884, 0.1288669073149633, 0.11969523249799581, 0.11554795361036506], Approach_calibrationAlpha=[1.5706246585230048, -8.758013512070892E-4, -0.018461075569511088, 1.5700128373526983, -1.56996879375117, 0.0], Approach_calibrationJointChecksum=[-1491211115, -1489904062, 825637646, -1324252155, -1324589245, -1493743004], Approach_calibrationStatus=2, Approach_calibrationValidChecksum=true, Approach_baseToFeature=[0.0, 0.0, 0.0, 0.0, 0.0, 0.0], Approach_TCPOffset=[-6.734893140250553E-6, -3.0887918176236706E-5, 1.0356231080421718E-5, 6.755448808060407E-5, -1.35938430410019E-5, -7.258580383443458E-6], Exit_calibrationDeltaTheta=[3.116151702300951E-8, 1.4166449605851306, 4.865070095092713, 0.0014795719880187595, -4.990860781074746E-7, -3.925871878279752E-8], Exit_calibrationA=[-1.0158439173703436E-5, -0.09403205366486023, -0.5713346358199152, 7.365520588418577E-5, -1.1425881794166018E-5, 0.0], Exit_calibrationD=[0.18077228301924886, -690.9574877576223, 691.0028500066884, 0.1288669073149633, 0.11969523249799581, 0.11554795361036506], Exit_calibrationAlpha=[1.5706246585230048, -8.758013512070892E-4, -0.018461075569511088, 1.5700128373526983, -1.56996879375117, 0.0], Exit_calibrationJointChecksum=[-1491211115, -1489904062, 825637646, -1324252155, -1324589245, -1493743004], Exit_calibrationStatus=2, Exit_calibrationValidChecksum=true, Exit_baseToFeature=[0.0, 0.0, 0.0, 0.0, 0.0, 0.0], Exit_TCPOffset=[-3.0497296392012485E-6, -6.69062324957781E-5, -3.013223529274578E-6, 1.2362428802079652E-4, 6.838395587397031E-6, -1.4326346248283778E-5], currentWizardState=LANDING, Pose(key=refBaseToFeature, Position(key=posePosition, Length(key=X value=0 unit=M), Length(key=Y value=0 unit=M), Length(key=Z value=0 unit=M)), Rotation(key=poseRotation, Angle(key=RX value=0 unit=RAD), Angle(key=RY value=0 unit=RAD), Angle(key=RZ value=0 unit=RAD))), Pose(key=refPose, Position(key=posePosition, Length(key=X value=0.367646 unit=M), Length(key=Y value=-0.129391 unit=M), Length(key=Z value=0.115026 unit=M)), Rotation(key=poseRotation, Angle(key=RX value=-2.216631 unit=RAD), Angle(key=RY value=-2.195355 unit=RAD), Angle(key=RZ value=-0.032926 unit=RAD))), JointPositions(key=Approach_jointpositions, JointPosition(key=[1], Angle(key=pos value=0.109921 unit=RAD)), JointPosition(key=[2], Angle(key=pos value=-1.905444 unit=RAD)), JointPosition(key=[3], Angle(key=pos value=-2.310368 unit=RAD)), JointPosition(key=[4], Angle(key=pos value=2.648518 unit=RAD)), JointPosition(key=[5], Angle(key=pos value=-1.593084 unit=RAD)), JointPosition(key=[6], Angle(key=pos value=0.104553 unit=RAD))), JointPositions(key=Exit_jointpositions, JointPosition(key=[1], Angle(key=pos value=0.109924 unit=RAD)), JointPosition(key=[2], Angle(key=pos value=-1.904189 unit=RAD)), JointPosition(key=[3], Angle(key=pos value=-2.310182 unit=RAD)), JointPosition(key=[4], Angle(key=pos value=2.647078 unit=RAD)), JointPosition(key=[5], Angle(key=pos value=-1.593062 unit=RAD)), JointPosition(key=[6], Angle(key=pos value=0.104568 unit=RAD))))
                URCap Generated Movements (polyscope-pallet-impl, Universal Robots) state(isChildrenLocked=true)
                  MoveL speed 250 mm/s, acceleration 1200 mm/s^2 (useActiveTCP=true) feature=referencePoin_2
                    Waypoint Approach_2: TCP in base x=367.615 y=-129.397 z=139.517 mm, rx=-2.2166 ry=-2.1953 rz=-0.0328 rad; joints [6.298, -109.175, -132.377, 151.748, -91.277, 5.99] deg; TCP offset x=0 y=0 z=0 mm, rx=0 ry=0 rz=0 rad; feature pose in base x=367.646 y=-129.391 z=115.026 mm, rx=-2.2166 ry=-2.1954 rz=-0.0329 rad
                  MoveL speed 250 mm/s, acceleration 1200 mm/s^2 (useActiveTCP=true) feature(featureName=referencePoin_2)
                    Waypoint ToolActionPoi_2: TCP in base x=367.646 y=-129.391 z=115.026 mm, rx=-2.2166 ry=-2.1954 rz=-0.0329 rad; joints [6.291, -111.972, -132.714, 154.886, -91.328, 5.96] deg; TCP offset x=0 y=0 z=0 mm, rx=0 ry=0 rz=0 rad
                  Folder Tool action
                    URCap RG Grip (OnRobot, OnRobot A/S) dataModel(rg-target-force=40.0, rg-target-width=0.1)
                  MoveL speed 250 mm/s, acceleration 1200 mm/s^2 (useActiveTCP=true) feature(featureName=referencePoin_2)
                    Waypoint Exit_3: TCP in base x=367.579 y=-129.393 z=140.171 mm, rx=-2.2165 ry=-2.1953 rz=-0.0328 rad; joints [6.299, -109.1, -132.37, 151.663, -91.277, 5.991] deg; TCP offset x=0 y=0 z=0 mm, rx=0 ry=0 rz=0 rad
    Waypoint hp: TCP in base x=292.997 y=15.071 z=398.72 mm, rx=2.2312 ry=-2.2053 rz=0.0033 rad; joints [39.465, -75.549, -131.57, -243.154, -90.002, -141.049] deg
  Halt
